# B&R Automation Studio project CleanChemi_SiteManagementSystem (part 3)

#### HA_DirSanitize.st
```iecst
(* Sanitizes File Device *)
FUNCTION_BLOCK HA_DirSanitize
	IF enable = FALSE THEN
		Internal.State										:= DIRSANITIZE_RESET;
	END_IF;

	CASE Internal.State OF
		DIRSANITIZE_RESET:
			status											:= 65534;
			brsmemset(ADR(Internal),0,SIZEOF(Internal));
			Internal.State									:= DIRSANITIZE_IDLE;
		DIRSANITIZE_IDLE:
			status											:= 65534;
			IF enable THEN
				IF pDevice <> 0 AND pDirDef <> 0 AND pFileList <> 0 THEN
					brsmemset(ADR(Internal),0,SIZEOF(Internal));
					status									:= 65535;
					Internal.State							:= DIRSANITIZE_EVALUATE_DIR;
				ELSE
					brsmemset(ADR(Internal),0,SIZEOF(Internal));
					status									:= 60001;
					Internal.State							:= DIRSANITIZE_ERROR;
				END_IF;
			END_IF;
		DIRSANITIZE_EVALUATE_DIR:
			status											:= 65535;
			// Determine DirIdx
			FOR Internal.i := 0 TO MAX_DIR_MAN_FILE_LIST_IDX DO
				brsmemcpy(ADR(Internal.FileListItem),pFileList+SIZEOF(Internal.FileListItem)*Internal.i,SIZEOF(Internal.FileListItem));
				IF Internal.FileListItem.Path = '' AND Internal.FileListItem.IsDir = FALSE THEN
					EXIT;
				ELSE
					Internal.Found 							:= FALSE;
					FOR Internal.j := 0 TO MAX_DIR_DEF_IDX DO
						brsmemcpy(ADR(Internal.DirDefItem),pDirDef+SIZEOF(Internal.DirDefItem)*Internal.j,SIZEOF(Internal.DirDefItem));
						IF Internal.DirDefItem.Valid THEN
							IF Internal.FileListItem.Path = Internal.DirDefItem.DirPath OR Internal.FileListItem.Path = '' THEN
								Internal.FileListItem.DirIdx := Internal.j;
								Internal.Found 				:= TRUE;
								EXIT;
							END_IF;
						END_IF;
					END_FOR;
					IF NOT Internal.Found THEN
						FOR Internal.j := MAX_DIR_DEF_IDX TO 0 BY -1 DO
							brsmemcpy(ADR(Internal.DirDefItem),pDirDef+SIZEOF(Internal.DirDefItem)*Internal.j,SIZEOF(Internal.DirDefItem));
							IF Internal.DirDefItem.Valid THEN
								Internal.Find := FIND(Internal.FileListItem.Path,Internal.DirDefItem.DirPath);
								IF Internal.Find <> 0 THEN
									Internal.TempPath := DELETE(Internal.FileListItem.Path,LEN(Internal.DirDefItem.DirPath),1);
									IF FIND(Internal.TempPath,'/') <> 0 OR Internal.DirDefItem.DirPath = '' THEN
										Internal.FileListItem.DirIdx := Internal.j;
										EXIT;
									END_IF;
								END_IF;
							END_IF;
						END_FOR;
					END_IF;
					brsmemcpy(pFileList+SIZEOF(Internal.FileListItem)*Internal.i,ADR(Internal.FileListItem),SIZEOF(Internal.FileListItem));
				END_IF;
			END_FOR;

			// Handle Directory Sanitation
			Internal.Found									:= FALSE;
			FOR Internal.i := 0 TO MAX_DIR_MAN_FILE_LIST_IDX DO
				brsmemcpy(ADR(Internal.FileListItem),pFileList+SIZEOF(Internal.FileListItem)*Internal.i,SIZEOF(Internal.FileListItem));
				IF Internal.FileListItem.Path = '' AND Internal.FileListItem.IsDir = FALSE THEN
					EXIT;
				ELSIF Internal.FileListItem.IsDir THEN
					brsmemcpy(ADR(Internal.DirDefItem),pDirDef+SIZEOF(Internal.DirDefItem)*Internal.FileListItem.DirIdx,SIZEOF(Internal.DirDefItem));
					IF NOT Internal.DirDefItem.Sanitize.AllowUndefinedDir AND Internal.DirDefItem.DirPath <> Internal.FileListItem.Path THEN
						Internal.Found					:= TRUE;
						Internal.FileListItem.Internal.1 := 1;
						brsmemcpy(pFileList+SIZEOF(Internal.FileListItem)*Internal.i,ADR(Internal.FileListItem),SIZEOF(Internal.FileListItem));
					END_IF;
				END_IF;
			END_FOR;
			Internal.State 									:= DIRSANITIZE_DELETE_DIR_CMD;
		DIRSANITIZE_DELETE_DIR_CMD:
			status											:= 65535;
			Internal.Found									:= FALSE;
			FOR Internal.i := 0 TO MAX_DIR_MAN_FILE_LIST_IDX DO
				brsmemcpy(ADR(Internal.FileListItem),pFileList+SIZEOF(Internal.FileListItem)*Internal.i,SIZEOF(Internal.FileListItem));
				IF Internal.FileListItem.Path = '' AND Internal.FileListItem.IsDir = FALSE THEN
					EXIT;
				ELSIF Internal.FileListItem.IsDir AND Internal.FileListItem.Internal.1 = 1 AND NOT Internal.FileListItem.Internal.2 = 1 THEN
					Internal.Found							:= TRUE;
					EXIT;
				END_IF;
			END_FOR;
			IF Internal.Found THEN
				Internal.DirDeleteEx_0.enable 				:= TRUE;
				Internal.DirDeleteEx_0.pDevice 				:= pDevice;
				Internal.DirDeleteEx_0.pName 				:= ADR(Internal.FileListItem.Path);
				Internal.State 								:= DIRSANITIZE_DELETE_DIR_WAIT;
			ELSE
				Internal.State 								:= DIRSANITIZE_EVALUATE_FILE;
			END_IF;
		DIRSANITIZE_DELETE_DIR_WAIT:
			status											:= 65535;
			IF Internal.DirDeleteEx_0.status = 0 OR (Internal.DirDeleteEx_0.status <> ERR_FUB_BUSY AND Internal.DirDeleteEx_0.status <> ERR_FUB_ENABLE_FALSE) THEN
				Internal.DirDeleteEx_0.enable 				:= FALSE;
				Internal.FileListItem1 						:= Internal.FileListItem;
				FOR Internal.i := 0 TO MAX_DIR_MAN_FILE_LIST_IDX DO
					brsmemcpy(ADR(Internal.FileListItem),pFileList+SIZEOF(Internal.FileListItem)*Internal.i,SIZEOF(Internal.FileListItem));
					IF Internal.FileListItem.Path = '' AND Internal.FileListItem.IsDir = FALSE THEN
						EXIT;
					ELSIF FIND(Internal.FileListItem.Path,Internal.FileListItem1.Path) <> 0 THEN
						Internal.FileListItem.Internal.3 	:= 1;
						brsmemcpy(pFileList+SIZEOF(Internal.FileListItem)*Internal.i,ADR(Internal.FileListItem),SIZEOF(Internal.FileListItem));
					END_IF;
				END_FOR;
				Internal.j 									:= 0;
				FOR Internal.i := 0 TO MAX_DIR_MAN_FILE_LIST_IDX DO
					brsmemcpy(ADR(Internal.FileListItem),pFileList+SIZEOF(Internal.FileListItem)*Internal.i,SIZEOF(Internal.FileListItem));
					IF Internal.FileListItem.Path = '' AND Internal.FileListItem.IsDir = FALSE THEN
						EXIT;
					ELSIF Internal.FileListItem.Internal.3 = 0 THEN
						IF Internal.j <> Internal.i THEN
							Internal.Size						:= (MAX_DIR_MAN_FILE_LIST_IDX+1-Internal.i);
							brsmemmove(pFileList+Internal.j*SIZEOF(Internal.FileListItem),pFileList+Internal.i*SIZEOF(Internal.FileListItem),SIZEOF(Internal.FileListItem)*Internal.Size);
							brsmemset(pFileList+(Internal.j+Internal.Size)*SIZEOF(Internal.FileListItem),0,SIZEOF(Internal.FileListItem)*(Internal.i-Internal.j));
						END_IF;
						Internal.j							:= Internal.j + (Internal.i-Internal.j)+1;
						Internal.i							:= Internal.j-1;
					ELSE
						brsmemset(pFileList+Internal.i*SIZEOF(Internal.FileListItem),0,SIZEOF(Internal.FileListItem));
					END_IF;
				END_FOR;
				Internal.State 								:= DIRSANITIZE_DELETE_DIR_CMD;
			END_IF;
		DIRSANITIZE_EVALUATE_FILE:
			status											:= 65535;

			// Handle File Sanitation By Root
			Internal.Found									:= FALSE;
			FOR Internal.i := 0 TO MAX_DIR_MAN_FILE_LIST_IDX DO
				brsmemcpy(ADR(Internal.FileListItem),pFileList+SIZEOF(Internal.FileListItem)*Internal.i,SIZEOF(Internal.FileListItem));
				IF Internal.FileListItem.Path = '' AND Internal.FileListItem.IsDir = FALSE THEN
					EXIT;
				ELSIF NOT Internal.FileListItem.IsDir THEN
					brsmemcpy(ADR(Internal.DirDefItem),pDirDef+SIZEOF(Internal.DirDefItem)*Internal.FileListItem.DirIdx,SIZEOF(Internal.DirDefItem));
					IF Internal.DirDefItem.Sanitize.SanitizeFilesByRoot THEN
						Internal.TempPath 					:= '';
						brsstrcat(ADR(Internal.TempPath),ADR(Internal.DirDefItem.DirPath));
						brsstrcat(ADR(Internal.TempPath),ADR('/'));
						brsstrcat(ADR(Internal.TempPath),ADR(Internal.DirDefItem.Sanitize.FileRoot));
						IF FIND(Internal.FileListItem.Path,Internal.TempPath) = 0 THEN
							Internal.Found					:= TRUE;
							Internal.FileListItem.Internal.1 := 1;
							brsmemcpy(pFileList+SIZEOF(Internal.FileListItem)*Internal.i,ADR(Internal.FileListItem),SIZEOF(Internal.FileListItem));
						END_IF;
					END_IF;
					IF Internal.DirDefItem.Sanitize.SanitizeFilesByExt THEN
						IF FIND(Internal.FileListItem.Path,Internal.DirDefItem.Sanitize.FileExtension) = 0 THEN
							Internal.Found					:= TRUE;
							Internal.FileListItem.Internal.1 := 1;
							brsmemcpy(pFileList+SIZEOF(Internal.FileListItem)*Internal.i,ADR(Internal.FileListItem),SIZEOF(Internal.FileListItem));
						END_IF;
					END_IF;
				END_IF;
			END_FOR;

			// Check if found in the last step. If so we have to go delete these files before counting them for size and number of files.
			IF Internal.Found THEN
				Internal.State 								:= DIRSANITIZE_DELETE_FILE_CMD;
			ELSE
				// Reorder Files for Evaluation
				FOR Internal.i := 0 TO MAX_DIR_MAN_FILE_LIST_IDX-1 DO
					brsmemcpy(ADR(Internal.FileListItem),pFileList+SIZEOF(Internal.FileListItem)*Internal.i,SIZEOF(Internal.FileListItem));
					brsmemcpy(ADR(Internal.FileListItem1),pFileList+SIZEOF(Internal.FileListItem1)*(Internal.i+1),SIZEOF(Internal.FileListItem1));
					IF (Internal.FileListItem.Path = '' AND Internal.FileListItem.IsDir = FALSE) OR (Internal.FileListItem1.Path = '' AND Internal.FileListItem1.IsDir = FALSE) THEN
						EXIT;
					ELSE
						IF Internal.FileListItem.DirIdx = Internal.FileListItem1.DirIdx THEN
							IF Internal.FileListItem.DateUDINT < Internal.FileListItem1.DateUDINT THEN
								brsmemcpy(pFileList+SIZEOF(Internal.FileListItem1)*Internal.i,ADR(Internal.FileListItem1),SIZEOF(Internal.FileListItem1));
								brsmemcpy(pFileList+SIZEOF(Internal.FileListItem)*(Internal.i+1),ADR(Internal.FileListItem),SIZEOF(Internal.FileListItem));
							END_IF;
						END_IF;
					END_IF;
				END_FOR;
				// Delete Files Based On File Number and Size Restriction
				Internal.Found								:= FALSE;
				Internal.CurrentDirIdx						:= 0;
				Internal.FileCount							:= 1;
				Internal.SizeCount							:= 0;
				FOR Internal.i := 0 TO MAX_DIR_MAN_FILE_LIST_IDX DO
					brsmemcpy(ADR(Internal.FileListItem),pFileList+SIZEOF(Internal.FileListItem)*Internal.i,SIZEOF(Internal.FileListItem));
					IF Internal.FileListItem.Path = '' AND Internal.FileListItem.IsDir = FALSE THEN
						EXIT;
					ELSIF NOT Internal.FileListItem.IsDir THEN
						IF Internal.CurrentDirIdx <> Internal.FileListItem.DirIdx THEN
							Internal.CurrentDirIdx 			:= Internal.FileListItem.DirIdx;
							Internal.FileCount				:= 1;
							Internal.SizeCount				:= Internal.FileListItem.Size;
						ELSE
							Internal.FileCount				:= Internal.FileCount + 1;
							Internal.SizeCount				:= Internal.SizeCount + Internal.FileListItem.Size;
						END_IF;
						brsmemcpy(ADR(Internal.DirDefItem),pDirDef+SIZEOF(Internal.DirDefItem)*Internal.FileListItem.DirIdx,SIZEOF(Internal.DirDefItem));
						IF Internal.FileCount > Internal.DirDefItem.Sanitize.MaxFiles OR Internal.SizeCount > Internal.DirDefItem.Sanitize.MaxSize THEN
							Internal.Found					:= TRUE;
							Internal.FileListItem.Internal.1 := 1;
							brsmemcpy(pFileList+SIZEOF(Internal.FileListItem)*Internal.i,ADR(Internal.FileListItem),SIZEOF(Internal.FileListItem));
						END_IF;
					END_IF;
				END_FOR;
				IF Internal.Found THEN
					Internal.State 							:= DIRSANITIZE_DELETE_FILE_CMD;
				ELSE
					Internal.State 							:= DIRSANITIZE_DONE;
				END_IF;
			END_IF;
		DIRSANITIZE_DELETE_FILE_CMD:
			status											:= 65535;
			Internal.Found									:= FALSE;
			FOR Internal.i := 0 TO MAX_DIR_MAN_FILE_LIST_IDX DO
				brsmemcpy(ADR(Internal.FileListItem),pFileList+SIZEOF(Internal.FileListItem)*Internal.i,SIZEOF(Internal.FileListItem));
				IF Internal.FileListItem.Path = '' AND Internal.FileListItem.IsDir = FALSE THEN
					EXIT;
				ELSIF NOT Internal.FileListItem.IsDir AND Internal.FileListItem.Internal.1 = 1 THEN
					Internal.FileListItem.Internal.1 := 0;
					Internal.FileListItem.Internal.3 := 1;
					brsmemcpy(pFileList+SIZEOF(Internal.FileListItem)*Internal.i,ADR(Internal.FileListItem),SIZEOF(Internal.FileListItem));
					Internal.Found							:= TRUE;
					EXIT;
				END_IF;
			END_FOR;
			IF Internal.Found THEN
				Internal.FileDelete_0.enable 				:= TRUE;
				Internal.FileDelete_0.pDevice 				:= pDevice;
				Internal.FileDelete_0.pName 				:= ADR(Internal.FileListItem.Path);
				Internal.State 								:= DIRSANITIZE_DELETE_FILE_WAIT;
			ELSE
				Internal.State 								:= DIRSANITIZE_EVALUATE_FILE;
			END_IF;
		DIRSANITIZE_DELETE_FILE_WAIT:
			status											:= 65535;
			IF Internal.FileDelete_0.status = 0 OR (Internal.FileDelete_0.status <> ERR_FUB_BUSY AND Internal.FileDelete_0.status <> ERR_FUB_ENABLE_FALSE) THEN
				Internal.FileDelete_0.enable 				:= FALSE;
				Internal.j 									:= 0;
				FOR Internal.i := 0 TO MAX_DIR_MAN_FILE_LIST_IDX DO
					brsmemcpy(ADR(Internal.FileListItem),pFileList+SIZEOF(Internal.FileListItem)*Internal.i,SIZEOF(Internal.FileListItem));
					IF Internal.FileListItem.Path = '' AND Internal.FileListItem.IsDir = FALSE THEN
						EXIT;
					ELSIF Internal.FileListItem.Internal.3 = 0 THEN
						IF Internal.j <> Internal.i THEN
							Internal.Size						:= (MAX_DIR_MAN_FILE_LIST_IDX+1-Internal.i);
							brsmemmove(pFileList+Internal.j*SIZEOF(Internal.FileListItem),pFileList+Internal.i*SIZEOF(Internal.FileListItem),SIZEOF(Internal.FileListItem)*Internal.Size);
							brsmemset(pFileList+(Internal.j+Internal.Size)*SIZEOF(Internal.FileListItem),0,SIZEOF(Internal.FileListItem)*(Internal.i-Internal.j));
						END_IF;
						Internal.j							:= Internal.j + (Internal.i-Internal.j)+1;
						Internal.i							:= Internal.j-1;
					ELSE
						brsmemset(pFileList+Internal.i*SIZEOF(Internal.FileListItem),0,SIZEOF(Internal.FileListItem));
					END_IF;
				END_FOR;
				Internal.State 								:= DIRSANITIZE_DELETE_FILE_CMD;
			END_IF;
		DIRSANITIZE_DONE:
			status											:= 0;
		DIRSANITIZE_ERROR:
			// Error
	END_CASE;

	Internal.FileDelete_0();
	Internal.DirDeleteEx_0();

END_FUNCTION_BLOCK
```

#### HA_Dir_USB_Connect.st
```iecst
// This function only supports a single USB flash drive, additional will be ignored.
// When connected the USB can be accessed using Dev Name 'USB_DEVICE'

FUNCTION_BLOCK HA_Dir_USB_Connect

	IF enable = FALSE OR reset THEN
		Internal.State											:= USB_CONNECT_RESET;
	END_IF;

	CASE Internal.State OF
		USB_CONNECT_RESET:
			status												:= 65534;
			brsmemset(ADR(Internal),0,SIZEOF(Internal));
			connected											:= FALSE;
			Internal.State										:= USB_CONNECT_IDLE;
		USB_CONNECT_IDLE:
			status												:= 65534;
			IF enable THEN
				status											:= 65535;
				Internal.State									:= USB_CONNECT_GET_LIST_CMD;
			END_IF;
		USB_CONNECT_GET_LIST_CMD:
			status												:= 65535;
			Internal.UsbNodeListGet_0.enable 					:= TRUE;
			Internal.UsbNodeListGet_0.pBuffer 					:= ADR(Internal.NodeList);
			Internal.UsbNodeListGet_0.bufferSize 				:= SIZEOF(Internal.NodeList);
			Internal.UsbNodeListGet_0.filterInterfaceClass 		:= 8; // FIND ONLY USB FLASH DRIVES
			Internal.UsbNodeListGet_0.filterInterfaceSubClass 	:= 6; // FIND ONLY USB FLASH DRIVES
			Internal.State 										:= USB_CONNECT_GET_LIST_WAIT;
		USB_CONNECT_GET_LIST_WAIT:
			status												:= 65535;
			IF Internal.UsbNodeListGet_0.status = 0 THEN
				Internal.UsbNodeListGet_0.enable 				:= FALSE;
				Internal.State 									:= USB_CONNECT_GET_NODE_CMD;
			ELSIF Internal.UsbNodeListGet_0.status <> ERR_FUB_BUSY AND Internal.UsbNodeListGet_0.status <> ERR_FUB_ENABLE_FALSE THEN
				IF Internal.UsbNodeListGet_0.status <> asusbERR_USB_NOTFOUND THEN
					Internal.UsbNodeListGet_0.enable 			:= FALSE;
					status										:= Internal.UsbNodeListGet_0.status;
					Internal.State 								:= USB_CONNECT_ERROR;
				ELSE
					Internal.UsbNodeListGet_0.enable 			:= FALSE;
					Internal.State 								:= USB_CONNECT_DELAY;
				END_IF;
			END_IF;
		USB_CONNECT_GET_NODE_CMD:
			status												:= 65535;
			Internal.UsbNodeGet_0.enable 						:= TRUE;
			Internal.UsbNodeGet_0.pBuffer 						:= ADR(Internal.Node);
			Internal.UsbNodeGet_0.bufferSize 					:= SIZEOF(Internal.Node);
			Internal.UsbNodeGet_0.nodeId 						:= Internal.NodeList;
			Internal.State 										:= USB_CONNECT_GET_NODE_WAIT;
		USB_CONNECT_GET_NODE_WAIT:
			status												:= 65535;
			IF Internal.UsbNodeGet_0.status = 0 THEN
				Internal.UsbNodeGet_0.enable 					:= FALSE;
				brsmemset(ADR(Internal.ParString),0,SIZEOF(Internal.ParString));
				brsstrcat(ADR(Internal.ParString),ADR('/DEVICE='));
				brsstrcat(ADR(Internal.ParString), ADR(Internal.Node.ifName));
				Internal.State 									:= USB_CONNECT_DEVLINK_CMD;
			ELSIF Internal.UsbNodeGet_0.status <> ERR_FUB_BUSY AND Internal.UsbNodeGet_0.status <> ERR_FUB_ENABLE_FALSE THEN
				IF Internal.UsbNodeGet_0.status <> asusbERR_USB_NOTFOUND THEN
					Internal.UsbNodeGet_0.enable 				:= FALSE;
					status										:= Internal.UsbNodeGet_0.status;
					Internal.State 								:= USB_CONNECT_ERROR;
				ELSE
					Internal.UsbNodeGet_0.enable 				:= FALSE;
					Internal.State 								:= USB_CONNECT_DELAY;
				END_IF;
			END_IF;
		USB_CONNECT_DEVLINK_CMD:
			status												:= 65535;
			Internal.DevLink_0.enable 							:= TRUE;
			Internal.DevLink_0.pDevice 							:= ADR('USB_DEVICE');
			Internal.DevLink_0.pParam 							:= ADR(Internal.ParString);
			Internal.State 										:= USB_CONNECT_DEVLINK_WAIT;
		USB_CONNECT_DEVLINK_WAIT:
			status												:= 65535;
			IF Internal.DevLink_0.status = 0 THEN
				Internal.DevLink_0.enable 						:= FALSE;
				Internal.Handle									:= Internal.DevLink_0.handle;
				connected										:= FALSE;
				Internal.State 									:= USB_CONNECT_CHECK_CONNECTED;
			ELSIF Internal.DevLink_0.status <> ERR_FUB_BUSY AND Internal.DevLink_0.status <> ERR_FUB_ENABLE_FALSE THEN
				Internal.DevLink_0.enable 						:= FALSE;
				Internal.State 									:= USB_CONNECT_DEVUNLINK_CMD;
			END_IF;
		USB_CONNECT_CHECK_CONNECTED:
			status												:= 65535;
			Internal.UsbMsDeviceReady_0.enable					:= TRUE;
			Internal.UsbMsDeviceReady_0.pIfName					:= ADR(Internal.Node.ifName);
			Internal.State 										:= USB_CONNECT_CONNECTED;
		USB_CONNECT_CONNECTED:
			status												:= 65535;
			IF Internal.UsbMsDeviceReady_0.status = 0 THEN
				connected										:= TRUE;
				Internal.UsbMsDeviceReady_0.enable 				:= FALSE;
				Internal.State 									:= USB_CONNECT_CHECK_CONNECTED;
			ELSIF Internal.UsbMsDeviceReady_0.status <> ERR_FUB_BUSY AND Internal.UsbMsDeviceReady_0.status <> ERR_FUB_ENABLE_FALSE THEN
				Internal.UsbMsDeviceReady_0.enable 				:= FALSE;
				Internal.State 									:= USB_CONNECT_DEVUNLINK_CMD;
			END_IF;
		USB_CONNECT_DEVUNLINK_CMD:
			status												:= 65535;
			Internal.DevUnlink_0.enable 						:= TRUE;
			Internal.DevUnlink_0.handle 						:= Internal.Handle;
			Internal.State 										:= USB_CONNECT_DEVUNLINK_WAIT;
		USB_CONNECT_DEVUNLINK_WAIT:
			status												:= 65535;
			IF Internal.DevUnlink_0.status = 0 OR (Internal.DevUnlink_0.status <> ERR_FUB_BUSY AND Internal.DevUnlink_0.status <> ERR_FUB_ENABLE_FALSE) THEN
				Internal.DevUnlink_0.enable 					:= FALSE;
				Internal.State 									:= USB_CONNECT_DELAY;
			END_IF;
		USB_CONNECT_DELAY:
			status												:= 65535;
			IF Internal.CTON_Delay.Q OR refresh THEN
				refresh 										:= FALSE;
				Internal.CTON_Delay(IN := FALSE);
				Internal.State 									:= USB_CONNECT_GET_LIST_CMD;
			ELSE
				Internal.CTON_Delay(IN := TRUE, PT := REAL_TO_TIME(delay*1000.0));
			END_IF;
 		USB_CONNECT_ERROR:
			connected 											:= FALSE;
	END_CASE;

	Internal.UsbNodeListGet_0();
	Internal.UsbNodeGet_0();
	Internal.DevLink_0();
	Internal.UsbMsDeviceReady_0();
	Internal.DevUnlink_0();

	IF connected THEN
		status													:= 0;
	END_IF;

END_FUNCTION_BLOCK
```

#### HA_Dir_Transfer.st
```iecst
(* Transfer List from Device to Another. Always Overwrites Existing. If either src or dest path includes directories, then the directories need to exist (this will not create them automatically) *)
FUNCTION_BLOCK HA_Dir_Transfer
	IF NOT enable THEN
		Internal.State 											:= TRANSFER_RESET;
	END_IF;

	CASE Internal.State OF
		TRANSFER_RESET:
			status												:= 65534;
			brsmemset(ADR(Internal),0,SIZEOF(Internal));
			Internal.State 										:= TRANSFER_IDLE;
		TRANSFER_IDLE:
			IF enable THEN
				IF pTransferList <> 0 THEN
					status										:= 65535;
					brsmemset(ADR(Internal),0,SIZEOF(Internal));
					Internal.ListIdx		 					:= 0;
					Internal.State 								:= TRANSFER_CHECK_LIST;
				ELSE
					status										:= 60001;
					Internal.State								:= TRANSFER_ERROR;
				END_IF;
			END_IF;
		TRANSFER_CHECK_LIST:
			status												:= 65535;
			IF Internal.ListIdx >= 0 AND Internal.ListIdx <= MAX_TRANSFER_LIST_IDX THEN
				brsmemcpy(ADR(Internal.TransferListItem),pTransferList+SIZEOF(Internal.TransferListItem)*Internal.ListIdx,SIZEOF(Internal.TransferListItem));
				IF Internal.TransferListItem.Valid THEN
					IF Internal.TransferListItem.SrcDelete AND Internal.TransferListItem.NoTransfer THEN
						IF Internal.TransferListItem.IsDir THEN
							Internal.State 						:= TRANSFER_DIR_DELETE_CMD;
						ELSE
							Internal.State 						:= TRANSFER_FILE_DELETE_CMD;
						END_IF;
					ELSIF Internal.TransferListItem.SrcCreateDir THEN
						Internal.State 							:= TRANSFER_DIR_CREATE_CMD;
					ELSIF Internal.TransferListItem.IsDir THEN
						Internal.State 							:= TRANSFER_DIR_COPY_CMD;
					ELSE
						Internal.State 							:= TRANSFER_FILE_COPY_CMD;
					END_IF;
				ELSE
					Internal.State 								:= TRANSFER_DONE;
				END_IF;
			ELSE
				Internal.State 									:= TRANSFER_DONE;
			END_IF;
		TRANSFER_DIR_COPY_CMD:
			status												:= 65535;
			Internal.DirCopy_0.enable 							:= TRUE;
			Internal.DirCopy_0.option 							:= fiOVERWRITE;
			Internal.DirCopy_0.pSrcDev 							:= ADR(Internal.TransferListItem.SrcDev);
			Internal.DirCopy_0.pSrcDir 							:= ADR(Internal.TransferListItem.SrcPath);
			Internal.DirCopy_0.pDestDev 						:= ADR(Internal.TransferListItem.DestDev);
			Internal.DirCopy_0.pDestDir 						:= ADR(Internal.TransferListItem.DestPath);
			Internal.State 										:= TRANSFER_DIR_COPY_WAIT;
		TRANSFER_DIR_COPY_WAIT:
			status												:= 65535;
			IF Internal.TransferListItem.SrcOrDestUSB AND NOT USB_Connected THEN
				Internal.DirCopy_0.enable 						:= FALSE;
				status											:= 65000;
				Internal.State 									:= TRANSFER_ERROR;
			ELSIF Internal.DirCopy_0.status = 0 THEN
				Internal.DirCopy_0.enable 						:= FALSE;
				IF Internal.TransferListItem.SrcDelete THEN
					Internal.State 								:= TRANSFER_DIR_DELETE_CMD;
				ELSE
					Internal.ListIdx							:= Internal.ListIdx + 1;
					Internal.State 								:= TRANSFER_CHECK_LIST;
				END_IF;
			ELSIF Internal.DirCopy_0.status <> ERR_FUB_BUSY AND Internal.DirCopy_0.status <> ERR_FUB_ENABLE_FALSE THEN
				Internal.DirCopy_0.enable 						:= FALSE;
				status											:= Internal.DirCopy_0.status;
				Internal.State 									:= TRANSFER_ERROR;
			END_IF;
		TRANSFER_DIR_DELETE_CMD:
			status												:= 65535;
			Internal.DirDeleteEx_0.enable 						:= TRUE;
			Internal.DirDeleteEx_0.pDevice 						:= ADR(Internal.TransferListItem.SrcDev);
			Internal.DirDeleteEx_0.pName	 					:= ADR(Internal.TransferListItem.SrcPath);
			Internal.State 										:= TRANSFER_DIR_DELETE_WAIT;
		TRANSFER_DIR_DELETE_WAIT:
			status												:= 65535;
			IF Internal.TransferListItem.SrcOrDestUSB AND NOT USB_Connected THEN
				Internal.DirDeleteEx_0.enable 					:= FALSE;
				status											:= 65000;
				Internal.State 									:= TRANSFER_ERROR;
			ELSIF Internal.DirDeleteEx_0.status = 0 THEN
				Internal.DirDeleteEx_0.enable 					:= FALSE;
				Internal.ListIdx								:= Internal.ListIdx + 1;
				Internal.State 									:= TRANSFER_CHECK_LIST;
			ELSIF Internal.DirDeleteEx_0.status <> ERR_FUB_BUSY AND Internal.DirDeleteEx_0.status <> ERR_FUB_ENABLE_FALSE THEN
				Internal.DirDeleteEx_0.enable 					:= FALSE;
				status											:= Internal.DirDeleteEx_0.status;
				Internal.State 									:= TRANSFER_ERROR;
			END_IF;
		TRANSFER_FILE_COPY_CMD:
			status												:= 65535;
			Internal.FileCopy_0.enable 							:= TRUE;
			Internal.FileCopy_0.option 							:= fiOVERWRITE;
			Internal.FileCopy_0.pSrcDev 						:= ADR(Internal.TransferListItem.SrcDev);
			Internal.FileCopy_0.pSrc	 						:= ADR(Internal.TransferListItem.SrcPath);
			Internal.FileCopy_0.pDestDev 						:= ADR(Internal.TransferListItem.DestDev);
			Internal.FileCopy_0.pDest							:= ADR(Internal.TransferListItem.DestPath);
			Internal.State 										:= TRANSFER_FILE_COPY_WAIT;
		TRANSFER_FILE_COPY_WAIT:
			status												:= 65535;
			IF Internal.TransferListItem.SrcOrDestUSB AND NOT USB_Connected THEN
				Internal.FileCopy_0.enable 						:= FALSE;
				status											:= 65000;
				Internal.State 									:= TRANSFER_ERROR;
			ELSIF Internal.FileCopy_0.status = 0 THEN
				Internal.FileCopy_0.enable 						:= FALSE;
				IF Internal.TransferListItem.SrcDelete THEN
					Internal.State 								:= TRANSFER_FILE_DELETE_CMD;
				ELSE
					Internal.ListIdx							:= Internal.ListIdx + 1;
					Internal.State 								:= TRANSFER_CHECK_LIST;
				END_IF;
			ELSIF Internal.FileCopy_0.status <> ERR_FUB_BUSY AND Internal.FileCopy_0.status <> ERR_FUB_ENABLE_FALSE THEN
				Internal.FileCopy_0.enable 						:= FALSE;
				status											:= Internal.FileCopy_0.status;
				Internal.State 									:= TRANSFER_ERROR;
			END_IF;
		TRANSFER_FILE_DELETE_CMD:
			status												:= 65535;
			Internal.FileDelete_0.enable 						:= TRUE;
			Internal.FileDelete_0.pDevice 						:= ADR(Internal.TransferListItem.SrcDev);
			Internal.FileDelete_0.pName	 						:= ADR(Internal.TransferListItem.SrcPath);
			Internal.State 										:= TRANSFER_FILE_DELETE_WAIT;
		TRANSFER_FILE_DELETE_WAIT:
			status												:= 65535;
			IF Internal.TransferListItem.SrcOrDestUSB AND NOT USB_Connected THEN
				Internal.FileDelete_0.enable 					:= FALSE;
				status											:= 65000;
				Internal.State 									:= TRANSFER_ERROR;
			ELSIF Internal.FileDelete_0.status = 0 THEN
				Internal.FileDelete_0.enable 					:= FALSE;
				Internal.ListIdx								:= Internal.ListIdx + 1;
				Internal.State 									:= TRANSFER_CHECK_LIST;
			ELSIF Internal.FileDelete_0.status <> ERR_FUB_BUSY AND Internal.FileDelete_0.status <> ERR_FUB_ENABLE_FALSE THEN
				Internal.FileDelete_0.enable 					:= FALSE;
				status											:= Internal.FileDelete_0.status;
				Internal.State 									:= TRANSFER_ERROR;
			END_IF;
		TRANSFER_DIR_CREATE_CMD:
			status												:= 65535;
			Internal.DirCreate_0.enable 						:= TRUE;
			Internal.DirCreate_0.pDevice 						:= ADR(Internal.TransferListItem.SrcDev);
			Internal.DirCreate_0.pName	 						:= ADR(Internal.TransferListItem.SrcPath);
			Internal.State 										:= TRANSFER_DIR_CREATE_WAIT;
		TRANSFER_DIR_CREATE_WAIT:
			status												:= 65535;
			IF Internal.TransferListItem.SrcOrDestUSB AND NOT USB_Connected THEN
				Internal.DirCreate_0.enable 					:= FALSE;
				status											:= 65000;
				Internal.State 									:= TRANSFER_ERROR;
			ELSIF Internal.DirCreate_0.status = 0 THEN
				Internal.DirCreate_0.enable 					:= FALSE;
				Internal.ListIdx								:= Internal.ListIdx + 1;
				Internal.State 									:= TRANSFER_CHECK_LIST;
			ELSIF Internal.DirCreate_0.status <> ERR_FUB_BUSY AND Internal.DirCreate_0.status <> ERR_FUB_ENABLE_FALSE THEN
				Internal.FileDelete_0.enable 					:= FALSE;
				status											:= Internal.DirCreate_0.status;
				Internal.State 									:= TRANSFER_ERROR;
			END_IF;
		TRANSFER_DONE:
			status												:= 0;
		TRANSFER_ERROR:
			// Error
	END_CASE;

	index 														:= Internal.ListIdx;

	Internal.DirCreate_0();
	Internal.DirCopy_0();
	Internal.FileCopy_0();
	Internal.DirDeleteEx_0();
	Internal.FileDelete_0();

END_FUNCTION_BLOCK
```

#### HA_DirReadAll.st
```iecst
(* Reads Entire File Device *)
FUNCTION_BLOCK HA_DirReadAll
	IF enable = FALSE THEN
		Internal.State														:= DIRREADALL_RESET;
	END_IF;

	CASE Internal.State OF
		DIRREADALL_RESET:
			status															:= 65534;
			brsmemset(ADR(Internal),0,SIZEOF(Internal));
			Internal.State													:= DIRREADALL_IDLE;
		DIRREADALL_IDLE:
			status															:= 65534;
			IF enable THEN
				IF pDevice <> 0 AND pFileList <> 0 THEN
					brsmemset(ADR(Internal),0,SIZEOF(Internal));
					brsmemset(pFileList,0,(SIZEOF(Internal.FileListItem)*(MAX_DIR_MAN_FILE_LIST_IDX+1)));
					Internal.FileListItem.DateUDINT := 0;
					Internal.FileListItem.IsDir := TRUE;
					Internal.FileListItem.Path := '';
					Internal.FileListItem.Size := 0;
					Internal.FileListItem.Internal.0 := 0;
					Internal.FileListIdx									:= 0;
					IF Internal.FileListIdx <= MAX_DIR_MAN_FILE_LIST_IDX THEN
						brsmemcpy(pFileList+SIZEOF(Internal.FileListItem)*Internal.FileListIdx,ADR(Internal.FileListItem),SIZEOF(Internal.FileListItem));
					END_IF;
					Internal.FileListIdx									:= Internal.FileListIdx + 1;
					status													:= 65535;
					Internal.CurrentDirPath									:= '';
					Internal.State											:= DIRREADALL_OPEN_CMD;
				ELSE
					brsmemset(ADR(Internal),0,SIZEOF(Internal));
					status													:= 60001;
					Internal.State											:= DIRREADALL_ERROR;
				END_IF;
			END_IF;
		DIRREADALL_OPEN_CMD:
			status															:= 65535;
			Internal.DirOpen_0.enable 										:= TRUE;
			Internal.DirOpen_0.pDevice 										:= pDevice;
			Internal.DirOpen_0.pName 										:= ADR(Internal.CurrentDirPath);
			Internal.State 													:= DIRREADALL_OPEN_WAIT;
		DIRREADALL_OPEN_WAIT:
			status															:= 65535;
			IF Internal.DirOpen_0.status = 0 THEN
				Internal.DirOpen_0.enable 									:= FALSE;
				Internal.DirIdent 											:= Internal.DirOpen_0.ident;
				Internal.State 												:= DIRREADALL_READ_CMD;
			ELSIF Internal.DirOpen_0.status <> ERR_FUB_BUSY AND Internal.DirOpen_0.status <> ERR_FUB_ENABLE_FALSE THEN
				Internal.DirOpen_0.enable 									:= FALSE;
				status														:= Internal.DirOpen_0.status;
				Internal.State 												:= DIRREADALL_ERROR;
			END_IF;
		DIRREADALL_READ_CMD:
			status															:= 65535;
			brsmemset(ADR(Internal.DirData),0,SIZEOF(Internal.DirData));
			Internal.DirReadEx_0.enable 									:= TRUE;
			Internal.DirReadEx_0.ident 										:= Internal.DirIdent;
			Internal.DirReadEx_0.pData 										:= ADR(Internal.DirData);
			Internal.DirReadEx_0.data_len 									:= SIZEOF(Internal.DirData);
			Internal.State 													:= DIRREADALL_READ_WAIT;
		DIRREADALL_READ_WAIT:
			status															:= 65535;
			IF Internal.DirReadEx_0.status = 0 THEN
				Internal.DirReadEx_0.enable 								:= FALSE;
				brsmemset(ADR(Internal.FileListItem),0,SIZEOF(Internal.FileListItem));
				IF Internal.DirData.Filename[0] <> 46 THEN // check for '.' or '..' and filter out, '.' is decimal 46 in ascii
					IF Internal.CurrentDirPath <> '' THEN
						brsstrcat(ADR(Internal.FileListItem.Path),ADR(Internal.CurrentDirPath));
						brsstrcat(ADR(Internal.FileListItem.Path),ADR('/'));
					END_IF;
					brsstrcat(ADR(Internal.FileListItem.Path),ADR(Internal.DirData.Filename));
					Internal.FileListItem.DateUDINT 						:= DT_TO_UDINT(Internal.DirData.Date);
					Internal.FileListItem.Size 								:= Internal.DirData.Filelength;
					Internal.FileListItem.IsDir 							:= Internal.DirData.Mode = 1;
					Internal.FileListItem.Internal.0						:= Internal.DirData.Mode = 1;
					IF Internal.FileListIdx >= MAX_DIR_MAN_FILE_LIST_IDX THEN
						Internal.State 										:= DIRREADALL_CLOSE_WAIT;
						Internal.DirClose_0.ident 							:= Internal.DirIdent;
						Internal.DirClose_0.enable 							:= TRUE;
					ELSE
						brsmemcpy(pFileList+SIZEOF(Internal.FileListItem)*Internal.FileListIdx,ADR(Internal.FileListItem),SIZEOF(Internal.FileListItem));
						Internal.FileListIdx								:= Internal.FileListIdx + 1;
						Internal.State 										:= DIRREADALL_READ_CMD;
					END_IF;
				ELSE
					Internal.State 											:= DIRREADALL_READ_CMD;
				END_IF;
			ELSIF Internal.DirReadEx_0.status <> ERR_FUB_BUSY AND Internal.DirReadEx_0.status <> ERR_FUB_ENABLE_FALSE THEN
				Internal.DirReadEx_0.enable 								:= FALSE;
				Internal.DirClose_0.ident 									:= Internal.DirIdent;
				Internal.DirClose_0.enable 									:= TRUE;
				Internal.State 												:= DIRREADALL_CLOSE_WAIT;
			END_IF;
		DIRREADALL_CLOSE_WAIT:
			status															:= 65535;
			IF Internal.DirClose_0.status = 0 OR (Internal.DirClose_0.status <> ERR_FUB_BUSY AND Internal.DirClose_0.status <> ERR_FUB_ENABLE_FALSE) THEN
				Internal.DirClose_0.enable 									:= FALSE;
				IF Internal.FileListIdx >= MAX_DIR_MAN_FILE_LIST_IDX THEN
					Internal.State 											:= DIRREADALL_EVALUATE;
				ELSE
					FOR Internal.i := 0 TO MAX_DIR_MAN_FILE_LIST_IDX DO
						brsmemcpy(ADR(Internal.FileListItem),pFileList+SIZEOF(Internal.FileListItem)*Internal.i,SIZEOF(Internal.FileListItem));
						IF Internal.FileListItem.Path = '' AND Internal.FileListItem.IsDir = FALSE THEN
							Internal.State 									:= DIRREADALL_EVALUATE;
							EXIT;
						ELSIF Internal.FileListItem.Internal.0 = 1 THEN
							Internal.CurrentDirPath							:= Internal.FileListItem.Path;
							Internal.FileListItem.Internal.0				:= 0;
							brsmemcpy(pFileList+SIZEOF(Internal.FileListItem)*Internal.i,ADR(Internal.FileListItem),SIZEOF(Internal.FileListItem));
							Internal.State 									:= DIRREADALL_OPEN_CMD;
							EXIT;
						END_IF;
					END_FOR;
				END_IF;
			END_IF;
		DIRREADALL_EVALUATE:
			status															:= 65535;
//			// Build Lists
//			FOR Internal.i := 0 TO MAX_DIR_MAN_FILE_LIST_IDX DO
//				IF Internal.FileList[Internal.i].Path = '' THEN
//					EXIT;
//				ELSIF Internal.FileList[Internal.i].IsDir THEN
//					FileList[Internal.FileListIdx] 							:= Internal.FileList[Internal.i];
//					IF Internal.FileListIdx < MAX_DIR_MAN_FILE_LIST_IDX THEN
//						Internal.FileListIdx								:= Internal.FileListIdx + 1;
//					END_IF;
//				ELSE
//					FileList[Internal.FileListIdx] 							:= Internal.FileList[Internal.i];
//					IF Internal.FileListIdx < MAX_DIR_MAN_FILE_LIST_IDX THEN
//						Internal.FileListIdx								:= Internal.FileListIdx + 1;
//					END_IF;
//				END_IF;
//			END_FOR;
//			FileList 														:= Internal.FileList;
//			Internal.FileListIdx 											:= 0;
			Internal.State 													:= DIRREADALL_DONE;
		DIRREADALL_DONE:
			status															:= 0;
		DIRREADALL_ERROR:
			// Error
	END_CASE;

	Internal.DirOpen_0();
	Internal.DirReadEx_0();
	Internal.DirClose_0();

END_FUNCTION_BLOCK
```

### Library Logical/Libraries/HA_Convert (IEC)

#### Types.typ - Exported data types
```iecst
TYPE
	HA_DT_Parser_Internal_typ : 	STRUCT
		DateTime : DATE_AND_TIME;
		dateTimeStruct : DTStructure;
		year : STRING[4];
		month : STRING[2];
		day : STRING[2];
		hour : STRING[2];
		minute : STRING[2];
		second : STRING[2];
	END_STRUCT;
	HA_DT_Formatter_Internal_typ : 	STRUCT
		dateTimeStruct : DTStructure;
		year : STRING[4];
		month : STRING[2];
		day : STRING[2];
		hour : STRING[2];
		minute : STRING[2];
		second : STRING[2];
		separator : STRING[1];
		c : USINT;
		i : UDINT;
		formatLen : UDINT;
		format : STRING[80];
		output : STRING[80];
		length : UDINT;
	END_STRUCT;
END_TYPE
```

#### HA_Convert.fun - Exported functions and function blocks
```iecst
FUNCTION HA_DT_Parser : BOOL
	VAR_INPUT
		pValueString : UDINT;
		pOutDT : UDINT;
	END_VAR
	VAR
		Internal : HA_DT_Parser_Internal_typ;
	END_VAR
END_FUNCTION

FUNCTION HA_DT_Formatter : BOOL
	VAR_INPUT
		value : DATE_AND_TIME;
		pInFormatString : UDINT; (*Optional*)
		pOutString : UDINT;
		OutStringLength : UDINT;
	END_VAR
	VAR
		Internal : HA_DT_Formatter_Internal_typ;
	END_VAR
END_FUNCTION
```

#### HA_DT_Formatter.st
```iecst
(* Formats DATE_AND_TIME Value into a string *)
FUNCTION HA_DT_Formatter
	HA_DT_Formatter 								:= TRUE;
	IF pOutString = 0 OR OutStringLength = 0 THEN
		HA_DT_Formatter 							:= FALSE;
	ELSE
		HA_DT_Formatter 							:= TRUE;
		Internal.output								:= '';
		Internal.formatLen 							:= brsstrlen(pInFormatString);
		IF pInFormatString = 0 OR Internal.formatLen = 0 OR Internal.formatLen > SIZEOF(Internal.format)-1 THEN
			Internal.format 						:= 'DT#y-m-d-h:M:s';
			Internal.formatLen 						:= brsstrlen(ADR(Internal.format));
		ELSE
			brsstrcpy(ADR(Internal.format),pInFormatString);
			Internal.formatLen 						:= brsstrlen(ADR(Internal.format));
		END_IF;
		DT_TO_DTStructure(value,ADR(Internal.dateTimeStruct));
		Internal.year 								:= UINT_TO_STRING(Internal.dateTimeStruct.year);
		Internal.month 								:= USINT_TO_STRING(Internal.dateTimeStruct.month);
		Internal.day 								:= USINT_TO_STRING(Internal.dateTimeStruct.day);
		Internal.hour 								:= USINT_TO_STRING(Internal.dateTimeStruct.hour);
		Internal.minute 							:= USINT_TO_STRING(Internal.dateTimeStruct.minute);
		Internal.second 							:= USINT_TO_STRING(Internal.dateTimeStruct.second);
		FOR Internal.i := 0 TO Internal.formatLen DO
			brsmemcpy(ADR(Internal.c),ADR(Internal.format)+Internal.i,1);
		    CASE Internal.c OF
		        121: //'y'
					IF Internal.length + 4 >= OutStringLength-1 THEN
						Internal.output 			:= '';
						HA_DT_Formatter 			:= FALSE;
						RETURN;
					ELSE
						Internal.length				:= brsstrcat(ADR(Internal.output),ADR(Internal.year)) - ADR(Internal.output);
					END_IF;
		        109: //'m'
					IF Internal.length + 2 >= OutStringLength-1 THEN
						Internal.output 			:= '';
						HA_DT_Formatter 			:= FALSE;
						RETURN;
					ELSE
						IF Internal.dateTimeStruct.month <= 9 THEN
							brsstrcat(ADR(Internal.output),ADR('0'));
						END_IF;
						Internal.length				:= brsstrcat(ADR(Internal.output),ADR(Internal.month)) - ADR(Internal.output);
					END_IF;
		        100: //'d'
					IF Internal.length + 2 >= OutStringLength-1 THEN
						Internal.output 			:= '';
						HA_DT_Formatter 			:= FALSE;
						RETURN;
					ELSE
						IF Internal.dateTimeStruct.day <= 9 THEN
							brsstrcat(ADR(Internal.output),ADR('0'));
						END_IF;
						Internal.length				:= brsstrcat(ADR(Internal.output),ADR(Internal.day)) - ADR(Internal.output);
					END_IF;
		        104: //'h'
					IF Internal.length + 2 >= OutStringLength-1 THEN
						Internal.output 			:= '';
						HA_DT_Formatter 			:= FALSE;
						RETURN;
					ELSE
						IF Internal.dateTimeStruct.hour <= 9 THEN
							brsstrcat(ADR(Internal.output),ADR('0'));
						END_IF;
						Internal.length				:= brsstrcat(ADR(Internal.output),ADR(Internal.hour)) - ADR(Internal.output);
					END_IF;
		        77: //'M'
					IF Internal.length + 2 >= OutStringLength-1 THEN
						Internal.output 			:= '';
						HA_DT_Formatter 			:= FALSE;
						RETURN;
					ELSE
						IF Internal.dateTimeStruct.minute <= 9 THEN
							brsstrcat(ADR(Internal.output),ADR('0'));
						END_IF;
						Internal.length				:= brsstrcat(ADR(Internal.output),ADR(Internal.minute)) - ADR(Internal.output);
					END_IF;
		        115: //'s'
					IF Internal.length + 2 >= OutStringLength-1 THEN
						Internal.output 			:= '';
						HA_DT_Formatter 			:= FALSE;
						RETURN;
					ELSE
						IF Internal.dateTimeStruct.second <= 9 THEN
							brsstrcat(ADR(Internal.output),ADR('0'));
						END_IF;
						Internal.length				:= brsstrcat(ADR(Internal.output),ADR(Internal.second)) - ADR(Internal.output);
					END_IF;
		        ELSE
					brsmemset(ADR(Internal.separator),0,SIZEOF(Internal.separator));
					brsmemcpy(ADR(Internal.separator),ADR(Internal.c),1);
					IF Internal.length + 1 >= OutStringLength-1 THEN
						Internal.output 			:= '';
						HA_DT_Formatter 			:= FALSE;
						RETURN;
					ELSE
						Internal.length				:= brsstrcat(ADR(Internal.output),ADR(Internal.separator)) - ADR(Internal.output);
					END_IF;
		    END_CASE
		END_FOR;
		IF NOT HA_DT_Formatter THEN
			brsmemset(pOutString,0,OutStringLength);
		ELSE
			brsstrcpy(pOutString,ADR(Internal.output));
		END_IF;
	END_IF;
END_FUNCTION
```

#### HA_DT_Parser.st
```iecst
(* Parses string into DATE_AND_TIME format !!!!!STRING MUST BE IN THE FORM OF DT#yyyy-mm-dd-hh:MM:ss!!!!! all other will fail*)
FUNCTION HA_DT_Parser
	HA_DT_Parser 						:= TRUE;
	IF pOutDT = 0 OR pValueString = 0 THEN
		HA_DT_Parser 					:= FALSE;
	ELSE
		HA_DT_Parser					:= TRUE;
		brsmemset(ADR(Internal),0,SIZEOF(Internal));
		brsmemcpy(ADR(Internal.year),pValueString+3,4);
		brsmemcpy(ADR(Internal.month),pValueString+8,2);
		brsmemcpy(ADR(Internal.day),pValueString+11,2);
		brsmemcpy(ADR(Internal.hour),pValueString+14,2);
		brsmemcpy(ADR(Internal.minute),pValueString+17,2);
		brsmemcpy(ADR(Internal.second),pValueString+20,2);
		Internal.dateTimeStruct.year	:= STRING_TO_UINT(Internal.year);
		Internal.dateTimeStruct.month	:= STRING_TO_USINT(Internal.month);
		Internal.dateTimeStruct.day		:= STRING_TO_USINT(Internal.day);
		Internal.dateTimeStruct.hour	:= STRING_TO_USINT(Internal.hour);
		Internal.dateTimeStruct.minute	:= STRING_TO_USINT(Internal.minute);
		Internal.dateTimeStruct.second	:= STRING_TO_USINT(Internal.second);
		Internal.DateTime := DTStructure_TO_DT(ADR(Internal.dateTimeStruct));
		brsmemcpy(pOutDT,ADR(Internal.DateTime),SIZEOF(Internal.DateTime));
	END_IF;
END_FUNCTION
```

### Library Logical/Libraries/HA_AlarmX (IEC)

#### Types.typ - Exported data types
```iecst
TYPE
	HA_AlarmX_Helper_Internal_typ : 	STRUCT
		Active : BOOL;
		AddText : STRING[1000];
		ArEventLogGetIdent_0 : ArEventLogGetIdent;
		ArEventLogWrite_0 : ArEventLogWrite;
	END_STRUCT;
	HA_ALARMX_ACTION_ENUM :
		(
		HA_ALARMX_ACTION_NONE,
		HA_ALARMX_ACTION_SET,
		HA_ALARMX_ACTION_SET_NO_LOG,
		HA_ALARMX_ACTION_ACK,
		HA_ALARMX_ACTION_ACK_NO_LOG,
		HA_ALARMX_ACTION_LOG_ONLY
		);
	HA_ALARMX_CORE_STATE_ENUM :
		(
		HA_ALARMX_CORE_RESET,
		HA_ALARMX_CORE_IDLE,
		HA_ALARMX_CORE_SET_C,
		HA_ALARMX_CORE_SET_W
		);
	HA_AlarmX_Core_Internal_typ : 	STRUCT
		state : HA_ALARMX_CORE_STATE_ENUM;
		currentAlarm : HA_AlarmX_Core_Buffer_typ;
		tDelay : CTON;
		i : INT;
	END_STRUCT;
	HA_AlarmX_Core_Buffer_typ : 	STRUCT
		name : STRING[MAX_ALARM_NAME_LEN];
		addText : ARRAY[0..HA_ALARMX_MAX_ADD_DATA_IDX]OF STRING[MAX_ALARM_ADD_DATA];
		allowMultiple : BOOL;
	END_STRUCT;
	HA_AlarmX_AlarmExtraData_typ : 	STRUCT
		AddData : ARRAY[0..HA_ALARMX_MAX_ADD_DATA_IDX]OF STRING[MAX_ALARM_ADD_DATA];
	END_STRUCT;
	HA_AlarmX_CfgMod_Internal_typ : 	STRUCT
		MpAlarmXConfigAlarm_0 : MpAlarmXConfigAlarm;
		AlarmCfg : MpAlarmXAlarmConfigType;
		AlarmName : STRING[MAX_ALARM_NAME_LEN];
		i : USINT;
		CTON_Timeout : CTON;
	END_STRUCT;
	HA_AlarmX_BufferInfo_typ : 	STRUCT
		Address : UDINT;
		Size : UDINT;
	END_STRUCT;
	HA_Module_Alarm_Info_typ : 	STRUCT
		ErrorInfo : USINT;
		IgnoreInfo : USINT;
	END_STRUCT;
END_TYPE
```

#### Constants.var - Exported constants
```iecst
VAR CONSTANT
	HA_MODULE_MAX_ALARM : USINT := 6;
	MAX_ALARM_ADD_DATA : UDINT := 255; (*Maximum Length of the extra alarm text*)
	MAX_ALARM_NAME_LEN : UDINT := 255; (*Maximum Length of the alarm name*)
	HA_ALARMX_BUFFER_IDX : UDINT := 255; (*Length of alarm buffer*)
	HA_ALARMX_MAX_ADD_DATA_IDX : USINT := 3;
END_VAR
```

#### HA_AlarmX.fun - Exported functions and function blocks
```iecst
{REDUND_ERROR} FUNCTION HA_AlarmX_Helper : DINT (*Helper Function for Setting and Acknowledging Alarms with User Logger support.*) (*$GROUP=User,$CAT=User,$GROUPICON=User.png,$CATICON=User.png*)
	VAR_INPUT
		MpLink : MpComIdentType;
		AlarmName : STRING[255];
		AlarmAction : HA_ALARMX_ACTION_ENUM;
		LogEventAddText : STRING[255];
		AllowMultiple : BOOL;
	END_VAR
	VAR
		Internal : HA_AlarmX_Helper_Internal_typ;
	END_VAR
END_FUNCTION

{REDUND_ERROR} FUNCTION_BLOCK HA_AlarmXCore (*TODO: Add your comment here*) (*$GROUP=User,$CAT=User,$GROUPICON=User.png,$CATICON=User.png*)
	VAR_INPUT
		enable : BOOL;
		MpLink : MpComIdentType;
		pBuffer : UDINT;
		pOutputData : REFERENCE TO HA_AlarmX_AlarmExtraData_typ;
		delayTime : TIME;
	END_VAR
	VAR
		internal : HA_AlarmX_Core_Internal_typ;
	END_VAR
END_FUNCTION_BLOCK

{REDUND_ERROR} {REDUND_UNREPLICABLE} FUNCTION_BLOCK HA_AlarmX_CfgModule (*Adds the HA default module alarms to the given alarmxcore*) (*$GROUP=User,$CAT=User,$GROUPICON=User.png,$CATICON=User.png*)
	VAR_INPUT
		MpLink : {REDUND_UNREPLICABLE} UDINT;
		Prefix : {REDUND_UNREPLICABLE} STRING[255];
		CodePrefix : {REDUND_UNREPLICABLE} UDINT;
	END_VAR
	VAR
		internal : {REDUND_UNREPLICABLE} HA_AlarmX_CfgMod_Internal_typ;
	END_VAR
	VAR_OUTPUT
		Error : BOOL;
	END_VAR
END_FUNCTION_BLOCK
```

#### HA_AlarmX_Helper.st
```iecst
(* Helper Function for Setting and Acknowledging Alarms with User Logger support. *)
FUNCTION HA_AlarmX_Helper
	HA_AlarmX_Helper 					:= -1;
	brsmemset(ADR(Internal),0,SIZEOF(Internal));
	Internal.ArEventLogGetIdent_0(Execute := FALSE);
	Internal.ArEventLogGetIdent_0(Execute := TRUE, Name := '$$arlogusr');
	Internal.AddText 					:= AlarmName;
	Internal.Active						:= NOT MpAlarmXCheckState(MpLink,AlarmName,mpALARMX_STATE_NONE);

	CASE AlarmAction OF
		HA_ALARMX_ACTION_NONE:
			HA_AlarmX_Helper 			:= 0;
		HA_ALARMX_ACTION_SET:
			HA_AlarmX_Helper 			:= 0;
			IF NOT Internal.Active OR AllowMultiple THEN
				MpAlarmXSet(MpLink,AlarmName);
				brsmemset(ADR(Internal.AddText),0,SIZEOF(Internal.AddText));
				Internal.AddText 	:= AlarmName;
				HA_brsstrcat(ADR(Internal.AddText),ADR(' - Set'),SIZEOF(Internal.AddText));
				IF LogEventAddText <> '' THEN
					HA_brsstrcat(ADR(Internal.AddText),ADR(' - Info: '),SIZEOF(Internal.AddText));
					HA_brsstrcat(ADR(Internal.AddText),ADR(LogEventAddText),SIZEOF(Internal.AddText));
				END_IF;
				Internal.ArEventLogWrite_0(Execute := FALSE);
				Internal.ArEventLogWrite_0(Execute := TRUE, Ident := Internal.ArEventLogGetIdent_0.Ident, EventID := -536870912, OriginRecordID := 0, ObjectID := 'HA_AlarmX_Helper', AddDataSize := brsstrlen(ADR(Internal.AddText)), AddDataFormat := 1, AddData := ADR(Internal.AddText), TimeStamp := 0);
			END_IF;
		HA_ALARMX_ACTION_SET_NO_LOG:
			HA_AlarmX_Helper 			:= 0;
			IF NOT Internal.Active OR AllowMultiple THEN
				MpAlarmXSet(MpLink,AlarmName);
				brsmemset(ADR(Internal.AddText),0,SIZEOF(Internal.AddText));
			END_IF;
		HA_ALARMX_ACTION_ACK:
			HA_AlarmX_Helper 			:= 0;
			IF Internal.Active THEN
				MpAlarmXAcknowledge(MpLink,AlarmName);
				brsmemset(ADR(Internal.AddText),0,SIZEOF(Internal.AddText));
				Internal.AddText 	:= AlarmName;
				HA_brsstrcat(ADR(Internal.AddText),ADR(' - Ack'),SIZEOF(Internal.AddText));
				IF LogEventAddText <> '' THEN
					HA_brsstrcat(ADR(Internal.AddText),ADR(' - Info: '),SIZEOF(Internal.AddText));
					HA_brsstrcat(ADR(Internal.AddText),ADR(LogEventAddText),SIZEOF(Internal.AddText));
				END_IF;
				Internal.ArEventLogWrite_0(Execute := FALSE);
				Internal.ArEventLogWrite_0(Execute := TRUE, Ident := Internal.ArEventLogGetIdent_0.Ident, EventID := -536870912, OriginRecordID := 0, ObjectID := 'HA_AlarmX_Helper', AddDataSize := brsstrlen(ADR(Internal.AddText)), AddDataFormat := 1, AddData := ADR(Internal.AddText), TimeStamp := 0);
			END_IF;
		HA_ALARMX_ACTION_ACK_NO_LOG:
			HA_AlarmX_Helper 			:= 0;
			IF Internal.Active THEN
				MpAlarmXAcknowledge(MpLink,AlarmName);
			END_IF;
		HA_ALARMX_ACTION_LOG_ONLY:
			HA_AlarmX_Helper 			:= 0;
			brsmemset(ADR(Internal.AddText),0,SIZEOF(Internal.AddText));
			IF LogEventAddText <> '' THEN
				HA_brsstrcat(ADR(Internal.AddText),ADR('Info: '),SIZEOF(Internal.AddText));
				HA_brsstrcat(ADR(Internal.AddText),ADR(LogEventAddText),SIZEOF(Internal.AddText));
				Internal.ArEventLogWrite_0(Execute := FALSE);
				Internal.ArEventLogWrite_0(Execute := TRUE, Ident := Internal.ArEventLogGetIdent_0.Ident, EventID := -536870912, OriginRecordID := 0, ObjectID := 'HA_AlarmX_Helper', AddDataSize := brsstrlen(ADR(Internal.AddText)), AddDataFormat := 1, AddData := ADR(Internal.AddText), TimeStamp := 0);
			END_IF;
	END_CASE;

END_FUNCTION
```

#### HA_AlarmXCore.st
```iecst
(* Alarm Core to handle setting multiple alarms in one cycle with different texts *)
FUNCTION_BLOCK HA_AlarmXCore

	IF enable = FALSE THEN
		internal.state := HA_ALARMX_CORE_RESET;
	END_IF

	CASE internal.state OF

		HA_ALARMX_CORE_RESET:

			brsmemset(ADR(internal.currentAlarm), 0, SIZEOF(internal.currentAlarm));
			internal.state := HA_ALARMX_CORE_IDLE;

		HA_ALARMX_CORE_IDLE:

			IF HA_Array_PeekBtm(pBuffer, SIZEOF(internal.currentAlarm) * HA_ALARMX_BUFFER_IDX, ADR(internal.currentAlarm), SIZEOF(internal.currentAlarm)) > 0 THEN
				HA_Array_Dequeue(pBuffer, SIZEOF(internal.currentAlarm) * HA_ALARMX_BUFFER_IDX, ADR(internal.currentAlarm), SIZEOF(internal.currentAlarm));
				internal.state := HA_ALARMX_CORE_SET_C;
			END_IF

		HA_ALARMX_CORE_SET_C:

			FOR internal.i := 0 TO HA_ALARMX_MAX_ADD_DATA_IDX DO
				pOutputData.AddData[internal.i]	:= internal.currentAlarm.addText[internal.i];
			END_FOR
			HA_AlarmX_Helper(MpLink, internal.currentAlarm.name, HA_ALARMX_ACTION_SET, '', internal.currentAlarm.allowMultiple);

			internal.state := HA_ALARMX_CORE_SET_W;

		HA_ALARMX_CORE_SET_W:

			internal.tDelay.IN	:= TRUE;
			internal.tDelay.PT	:= delayTime;

			IF internal.tDelay.Q THEN
				internal.tDelay.IN	:= FALSE;
				internal.state 		:= HA_ALARMX_CORE_IDLE;
			END_IF

	END_CASE

	internal.tDelay();

END_FUNCTION_BLOCK
```

#### HA_AlarmX_CfgModule.st
```iecst
(* Adds the HA default module alarms to the given alarmxcore *)
FUNCTION_BLOCK HA_AlarmX_CfgModule

	WHILE internal.i < HA_MODULE_MAX_ALARM + 1 DO

		CASE internal.i OF

			0:
				internal.AlarmName														:= Prefix;
				HA_brsstrcat(ADR(internal.AlarmName), ADR('UnhandledCmd'), SIZEOF(internal.AlarmName));
				internal.AlarmCfg.Message												:= '{$$IAT/Alarm.';
				HA_brsstrcat(ADR(internal.AlarmCfg.Message), ADR(internal.AlarmName), SIZEOF(internal.AlarmCfg.Message));
				HA_brsstrcat(ADR(internal.AlarmCfg.Message), ADR('}'), SIZEOF(internal.AlarmCfg.Message));
				internal.AlarmCfg.Code													:= CodePrefix;
				internal.AlarmCfg.Severity												:= 4;
				internal.AlarmCfg.Behavior.AutoReset									:= TRUE;
				internal.AlarmCfg.Behavior.Acknowledge 									:= mpALARMX_ACK_REQ;
				internal.AlarmCfg.Behavior.MultipleInstances 							:= TRUE;
				internal.AlarmCfg.Behavior.ReactionUntilAcknowledged					:= TRUE;
				internal.AlarmCfg.Behavior.HistoryReport.InactiveToActive 				:= TRUE;
				internal.AlarmCfg.Behavior.HistoryReport.UnacknowledgedToAcknowledged	:= TRUE;

			1:
				internal.AlarmName															:= Prefix;
				HA_brsstrcat(ADR(internal.AlarmName), ADR('Severity1'), SIZEOF(internal.AlarmName));
				internal.AlarmCfg.Message												:= '{$$IAT/Alarm.';
				HA_brsstrcat(ADR(internal.AlarmCfg.Message), ADR('Severity1'), SIZEOF(internal.AlarmCfg.Message));
				HA_brsstrcat(ADR(internal.AlarmCfg.Message), ADR('}'), SIZEOF(internal.AlarmCfg.Message));
				internal.AlarmCfg.Code													:= CodePrefix;
				internal.AlarmCfg.Severity												:= 1;
				internal.AlarmCfg.Behavior.AutoReset									:= TRUE;
				internal.AlarmCfg.Behavior.Acknowledge 									:= mpALARMX_ACK_REQ;
				internal.AlarmCfg.Behavior.MultipleInstances 							:= TRUE;
				internal.AlarmCfg.Behavior.ReactionUntilAcknowledged					:= TRUE;
				internal.AlarmCfg.Behavior.HistoryReport.InactiveToActive 				:= TRUE;
				internal.AlarmCfg.Behavior.HistoryReport.UnacknowledgedToAcknowledged	:= TRUE;

			2:
				internal.AlarmName															:= Prefix;
				HA_brsstrcat(ADR(internal.AlarmName), ADR('Severity2'), SIZEOF(internal.AlarmName));
				internal.AlarmCfg.Message												:= '{$$IAT/Alarm.';
				HA_brsstrcat(ADR(internal.AlarmCfg.Message), ADR('Severity2'), SIZEOF(internal.AlarmCfg.Message));
				HA_brsstrcat(ADR(internal.AlarmCfg.Message), ADR('}'), SIZEOF(internal.AlarmCfg.Message));
				internal.AlarmCfg.Code													:= CodePrefix;
				internal.AlarmCfg.Severity												:= 2;
				internal.AlarmCfg.Behavior.AutoReset									:= TRUE;
				internal.AlarmCfg.Behavior.Acknowledge 									:= mpALARMX_ACK_REQ;
				internal.AlarmCfg.Behavior.MultipleInstances 							:= TRUE;
				internal.AlarmCfg.Behavior.ReactionUntilAcknowledged					:= TRUE;
				internal.AlarmCfg.Behavior.HistoryReport.InactiveToActive 				:= TRUE;
				internal.AlarmCfg.Behavior.HistoryReport.UnacknowledgedToAcknowledged	:= TRUE;

			3:
				internal.AlarmName															:= Prefix;
				HA_brsstrcat(ADR(internal.AlarmName), ADR('Severity3'), SIZEOF(internal.AlarmName));
				internal.AlarmCfg.Message												:= '{$$IAT/Alarm.';
				HA_brsstrcat(ADR(internal.AlarmCfg.Message), ADR('Severity3'), SIZEOF(internal.AlarmCfg.Message));
				HA_brsstrcat(ADR(internal.AlarmCfg.Message), ADR('}'), SIZEOF(internal.AlarmCfg.Message));
				internal.AlarmCfg.Code													:= CodePrefix;
				internal.AlarmCfg.Severity												:= 3;
				internal.AlarmCfg.Behavior.AutoReset									:= TRUE;
				internal.AlarmCfg.Behavior.Acknowledge 									:= mpALARMX_ACK_REQ;
				internal.AlarmCfg.Behavior.MultipleInstances 							:= TRUE;
				internal.AlarmCfg.Behavior.ReactionUntilAcknowledged					:= TRUE;
				internal.AlarmCfg.Behavior.HistoryReport.InactiveToActive 				:= TRUE;
				internal.AlarmCfg.Behavior.HistoryReport.UnacknowledgedToAcknowledged	:= TRUE;

			4:
				internal.AlarmName															:= Prefix;
				HA_brsstrcat(ADR(internal.AlarmName), ADR('Severity4'), SIZEOF(internal.AlarmName));
				internal.AlarmCfg.Message												:= '{$$IAT/Alarm.';
				HA_brsstrcat(ADR(internal.AlarmCfg.Message), ADR('Severity4'), SIZEOF(internal.AlarmCfg.Message));
				HA_brsstrcat(ADR(internal.AlarmCfg.Message), ADR('}'), SIZEOF(internal.AlarmCfg.Message));
				internal.AlarmCfg.Code													:= CodePrefix;
				internal.AlarmCfg.Severity												:= 4;
				internal.AlarmCfg.Behavior.AutoReset									:= TRUE;
				internal.AlarmCfg.Behavior.Acknowledge 									:= mpALARMX_ACK_REQ;
				internal.AlarmCfg.Behavior.MultipleInstances 							:= TRUE;
				internal.AlarmCfg.Behavior.ReactionUntilAcknowledged					:= TRUE;
				internal.AlarmCfg.Behavior.HistoryReport.InactiveToActive 				:= TRUE;
				internal.AlarmCfg.Behavior.HistoryReport.UnacknowledgedToAcknowledged	:= TRUE;

			5:
				internal.AlarmName															:= Prefix;
				HA_brsstrcat(ADR(internal.AlarmName), ADR('Severity5'), SIZEOF(internal.AlarmName));
				internal.AlarmCfg.Message												:= '{$$IAT/Alarm.';
				HA_brsstrcat(ADR(internal.AlarmCfg.Message), ADR('Severity5'), SIZEOF(internal.AlarmCfg.Message));
				HA_brsstrcat(ADR(internal.AlarmCfg.Message), ADR('}'), SIZEOF(internal.AlarmCfg.Message));
				internal.AlarmCfg.Code													:= CodePrefix;
				internal.AlarmCfg.Severity												:= 5;
				internal.AlarmCfg.Behavior.AutoReset									:= TRUE;
				internal.AlarmCfg.Behavior.Acknowledge 									:= mpALARMX_ACK_REQ;
				internal.AlarmCfg.Behavior.MultipleInstances 							:= TRUE;
				internal.AlarmCfg.Behavior.ReactionUntilAcknowledged					:= TRUE;
				internal.AlarmCfg.Behavior.HistoryReport.InactiveToActive 				:= TRUE;
				internal.AlarmCfg.Behavior.HistoryReport.UnacknowledgedToAcknowledged	:= TRUE;

			6:
				internal.AlarmName														:= Prefix;
				HA_brsstrcat(ADR(internal.AlarmName), ADR('CmdIgnored'), SIZEOF(internal.AlarmName));
				internal.AlarmCfg.Message												:= '{$$IAT/Alarm.';
				HA_brsstrcat(ADR(internal.AlarmCfg.Message), ADR(internal.AlarmName), SIZEOF(internal.AlarmCfg.Message));
				HA_brsstrcat(ADR(internal.AlarmCfg.Message), ADR('}'), SIZEOF(internal.AlarmCfg.Message));
				internal.AlarmCfg.Code													:= CodePrefix + 6;
				internal.AlarmCfg.Severity												:= 0;
				internal.AlarmCfg.Behavior.AutoReset									:= TRUE;
				internal.AlarmCfg.Behavior.Acknowledge 									:= mpALARMX_ACK_REQ;
				internal.AlarmCfg.Behavior.MultipleInstances 							:= TRUE;
				internal.AlarmCfg.Behavior.ReactionUntilAcknowledged					:= TRUE;
				internal.AlarmCfg.Behavior.HistoryReport.InactiveToActive 				:= TRUE;
				internal.AlarmCfg.Behavior.HistoryReport.UnacknowledgedToAcknowledged	:= TRUE;

		END_CASE

		internal.MpAlarmXConfigAlarm_0.MpLink			:= MpLink;
		internal.MpAlarmXConfigAlarm_0.Enable			:= TRUE;
		internal.MpAlarmXConfigAlarm_0.Name				:= ADR(internal.AlarmName);
		internal.MpAlarmXConfigAlarm_0.Configuration	:= ADR(internal.AlarmCfg);
		internal.MpAlarmXConfigAlarm_0.Save				:= TRUE;

		IF internal.MpAlarmXConfigAlarm_0.CommandDone THEN
			internal.i := internal.i + 1;
			internal.MpAlarmXConfigAlarm_0.Save := FALSE;
		ELSIF internal.MpAlarmXConfigAlarm_0.Error THEN
			Error	:= TRUE;
			RETURN;
		END_IF;

		internal.MpAlarmXConfigAlarm_0();
	END_WHILE

END_FUNCTION_BLOCK
```

### Library Logical/Libraries/HA_ItemX (IEC)

#### Types.typ - Exported data types
```iecst
TYPE
	ItemX_typ : 	STRUCT
		CurrentUID : UDINT; (*REQUIRED*)
		ValidIndex : BOOL; (*REQUIRED*)
		ReturnedIndex : INT; (*REQUIRED*)
		Elem : ItemX_Elem_typ; (*REQUIRED*)
		List : ARRAY[0..MAX_ITEM_X_IDX]OF ItemX_Elem_typ; (*REQUIRED*)
	END_STRUCT;
	ItemX_Elem_typ : 	STRUCT
		UID : UDINT; (*REQUIRED*)
		State : ITEM_X_STATE_ENUM; (*REQUIRED*)
		LastLoc : ITEM_X_LOC_ENUM; (*REQUIRED*)
		Loc : ITEM_X_LOC_ENUM; (*REQUIRED*)
		Par : ItemX_Par_typ; (*REQUIRED*)
		Status : ItemX_Status_typ; (*REQUIRED*)
	END_STRUCT;
	ItemX_Status_typ : 	STRUCT
		Position : REAL;
		Length : REAL;
		ManuallyRemoved : BOOL;
		Rejected : BOOL;
		Passed : BOOL;
		TimeIn : DATE_AND_TIME;
		TimeOut : DATE_AND_TIME;
		Error : BOOL;
	END_STRUCT;
	ItemX_Par_typ : 	STRUCT
		ProductID : INT;
		Recipe : ItemX_Par_Recipe_typ;
	END_STRUCT;
	ItemX_Par_Recipe_typ : 	STRUCT
		MaxLength : REAL;
	END_STRUCT;
	ITEM_X_STATE_ENUM :
		(
		ITEM_X_STATE_UNDEFINED, (*REQUIRED*)
		ITEM_X_STATE_WAIT_START,
		ITEM_X_STATE_ACTIVE,
		ITEM_X_STATE_DONE,
		ITEM_X_STATE_UNKNOWN,
		ITEM_X_STATE_ERRORSTOP
		);
	ITEM_X_LOC_ENUM :
		(
		ITEM_X_LOC_UNDEFINED, (*REQUIRED*)
		ITEM_X_LOC_UNKNOWN
		);
	HA_ItemX_Internal_typ : 	STRUCT
		i : INT;
		j : INT;
		tempItemX : ItemX_Elem_typ;
		tempIndex : INT;
		tempUID : UDINT;
	END_STRUCT;
END_TYPE
```

#### Constants.var - Exported constants
```iecst
VAR CONSTANT
	MAX_ITEM_X_IDX : INT := 15;
	MAX_NAME_STRING_LENGTH : INT := 30;
END_VAR
```

#### HA_ItemX.fun - Exported functions and function blocks
```iecst
{REDUND_ERROR} FUNCTION HA_ItemX_DeleteByIndex : BOOL (* *) (*$GROUP=User,$CAT=User,$GROUPICON=User.png,$CATICON=User.png*)
	VAR_INPUT
		Index : INT;
	END_VAR
	VAR_IN_OUT
		ItemX : ItemX_typ;
	END_VAR
	VAR
		Internal : HA_ItemX_Internal_typ;
	END_VAR
END_FUNCTION

{REDUND_ERROR} FUNCTION HA_ItemX_DeleteByUID : BOOL (* *) (*$GROUP=User,$CAT=User,$GROUPICON=User.png,$CATICON=User.png*)
	VAR_INPUT
		UID : UDINT;
	END_VAR
	VAR_IN_OUT
		ItemX : ItemX_typ;
	END_VAR
	VAR
		Internal : HA_ItemX_Internal_typ;
	END_VAR
END_FUNCTION

{REDUND_ERROR} FUNCTION HA_ItemX_UID_TO_Index : BOOL (* *) (*$GROUP=User,$CAT=User,$GROUPICON=User.png,$CATICON=User.png*)
	VAR_INPUT
		UID : UDINT;
	END_VAR
	VAR_IN_OUT
		ItemX : ItemX_typ;
	END_VAR
	VAR
		Internal : HA_ItemX_Internal_typ;
	END_VAR
END_FUNCTION

{REDUND_ERROR} FUNCTION HA_ItemX_Sanitize : BOOL (* *) (*$GROUP=User,$CAT=User,$GROUPICON=User.png,$CATICON=User.png*)
	VAR_IN_OUT
		ItemX : ItemX_typ;
	END_VAR
	VAR
		Internal : HA_ItemX_Internal_typ;
	END_VAR
END_FUNCTION

{REDUND_ERROR} FUNCTION HA_ItemX_Reorder_LowToHighUID : BOOL (* *) (*$GROUP=User,$CAT=User,$GROUPICON=User.png,$CATICON=User.png*)
	VAR_IN_OUT
		ItemX : ItemX_typ;
	END_VAR
	VAR
		Internal : HA_ItemX_Internal_typ;
	END_VAR
END_FUNCTION

{REDUND_ERROR} FUNCTION HA_ItemX_Reorder_HighToLowUID : BOOL (* *) (*$GROUP=User,$CAT=User,$GROUPICON=User.png,$CATICON=User.png*)
	VAR_IN_OUT
		ItemX : ItemX_typ;
	END_VAR
	VAR
		Internal : HA_ItemX_Internal_typ;
	END_VAR
END_FUNCTION

{REDUND_ERROR} FUNCTION HA_ItemX_IndexLowestUID : BOOL (* *) (*$GROUP=User,$CAT=User,$GROUPICON=User.png,$CATICON=User.png*)
	VAR_IN_OUT
		ItemX : ItemX_typ;
	END_VAR
	VAR
		Internal : HA_ItemX_Internal_typ;
	END_VAR
END_FUNCTION

{REDUND_ERROR} FUNCTION HA_ItemX_IndexHighestUID : BOOL (* *) (*$GROUP=User,$CAT=User,$GROUPICON=User.png,$CATICON=User.png*)
	VAR_IN_OUT
		ItemX : ItemX_typ;
	END_VAR
	VAR
		Internal : HA_ItemX_Internal_typ;
	END_VAR
END_FUNCTION

{REDUND_ERROR} FUNCTION HA_ItemX_FirstOpenIndex : BOOL (* *) (*$GROUP=User,$CAT=User,$GROUPICON=User.png,$CATICON=User.png*)
	VAR_IN_OUT
		ItemX : ItemX_typ;
	END_VAR
	VAR
		Internal : HA_ItemX_Internal_typ;
	END_VAR
END_FUNCTION

{REDUND_ERROR} FUNCTION HA_ItemX_GetElemByIndex : BOOL (* *) (*$GROUP=User,$CAT=User,$GROUPICON=User.png,$CATICON=User.png*)
	VAR_INPUT
		Index : INT;
	END_VAR
	VAR_IN_OUT
		ItemX : ItemX_typ;
	END_VAR
	VAR
		Internal : HA_ItemX_Internal_typ;
	END_VAR
END_FUNCTION

{REDUND_ERROR} FUNCTION HA_ItemX_GetElemByUID : BOOL (* *) (*$GROUP=User,$CAT=User,$GROUPICON=User.png,$CATICON=User.png*)
	VAR_INPUT
		UID : UDINT;
	END_VAR
	VAR_IN_OUT
		ItemX : ItemX_typ;
	END_VAR
	VAR
		Internal : HA_ItemX_Internal_typ;
	END_VAR
END_FUNCTION

{REDUND_ERROR} FUNCTION HA_ItemX_ModElemByIndex : BOOL (* *) (*$GROUP=User,$CAT=User,$GROUPICON=User.png,$CATICON=User.png*)
	VAR_INPUT
		Index : INT;
	END_VAR
	VAR_IN_OUT
		ItemX : ItemX_typ;
	END_VAR
	VAR
		Internal : HA_ItemX_Internal_typ;
	END_VAR
END_FUNCTION

{REDUND_ERROR} FUNCTION HA_ItemX_ModElemByUID : BOOL (* *) (*$GROUP=User,$CAT=User,$GROUPICON=User.png,$CATICON=User.png*)
	VAR_INPUT
		UID : UDINT;
	END_VAR
	VAR_IN_OUT
		ItemX : ItemX_typ;
	END_VAR
	VAR
		Internal : HA_ItemX_Internal_typ;
	END_VAR
END_FUNCTION

{REDUND_ERROR} FUNCTION HA_ItemX_AddElem : BOOL (* *) (*$GROUP=User,$CAT=User,$GROUPICON=User.png,$CATICON=User.png*)
	VAR_IN_OUT
		ItemX : ItemX_typ;
	END_VAR
	VAR
		Internal : HA_ItemX_Internal_typ;
	END_VAR
END_FUNCTION

{REDUND_ERROR} FUNCTION HA_ItemX_IncrementUID : BOOL (* *) (*$GROUP=User,$CAT=User,$GROUPICON=User.png,$CATICON=User.png*)
	VAR_IN_OUT
		ItemX : ItemX_typ;
	END_VAR
	VAR
		Internal : HA_ItemX_Internal_typ;
	END_VAR
END_FUNCTION
```

#### HA_ItemX_FirstOpenIndex.st
```iecst
(* Finds the first open index of the item array *)
FUNCTION HA_ItemX_FirstOpenIndex
	HA_ItemX_FirstOpenIndex							:= FALSE;
	ItemX.ReturnedIndex								:= -1;
	FOR Internal.i := 0 TO MAX_ITEM_X_IDX DO
		IF ItemX.List[Internal.i].UID = 0 THEN
			HA_ItemX_FirstOpenIndex					:= TRUE;
			ItemX.ReturnedIndex						:= Internal.i;
			EXIT;
		END_IF;
	END_FOR;

	// This is here for keeping the ItemX structure up to date and should be at the bottom of every function call in the library
	ItemX.ValidIndex									:= FALSE;
	IF ItemX.ReturnedIndex >= 0 AND ItemX.ReturnedIndex <= MAX_ITEM_X_IDX THEN
		ItemX.ValidIndex								:= TRUE;
	END_IF;

END_FUNCTION
```

#### HA_ItemX_UID_TO_Index.st
```iecst
(* Returns the first index matching the UID entered *)
FUNCTION HA_ItemX_UID_TO_Index
	HA_ItemX_UID_TO_Index							:= FALSE;
	ItemX.ReturnedIndex								:= -1;
	FOR Internal.i := 0 TO MAX_ITEM_X_IDX DO
		IF ItemX.List[Internal.i].UID = UID THEN
			HA_ItemX_UID_TO_Index					:= TRUE;
			ItemX.ReturnedIndex						:= Internal.i;
			EXIT;
		END_IF;
	END_FOR;

	// This is here for keeping the ItemX structure up to date and should be at the bottom of every function call in the library
	ItemX.ValidIndex									:= FALSE;
	IF ItemX.ReturnedIndex >= 0 AND ItemX.ReturnedIndex <= MAX_ITEM_X_IDX THEN
		ItemX.ValidIndex								:= TRUE;
	END_IF;

END_FUNCTION
```

#### HA_ItemX_DeleteByUID.st
```iecst
(* Deletes the first index matching the UID entered, Returns True if Deleted, False if not found *)
FUNCTION HA_ItemX_DeleteByUID
	HA_ItemX_DeleteByUID								:= FALSE;
	ItemX.ReturnedIndex								:= -1;
	FOR Internal.i := 0 TO MAX_ITEM_X_IDX DO
		IF ItemX.List[Internal.i].UID = UID THEN
			brsmemset(ADR(ItemX.List[Internal.i]),0,SIZEOF(ItemX.List[Internal.i]));
			ItemX.ReturnedIndex						:= Internal.i;
			HA_ItemX_DeleteByUID						:= TRUE;
			EXIT;
		END_IF;
	END_FOR;

	// This is here for keeping the ItemX structure up to date and should be at the bottom of every function call in the library
	ItemX.ValidIndex									:= FALSE;
	IF ItemX.ReturnedIndex >= 0 AND ItemX.ReturnedIndex <= MAX_ITEM_X_IDX THEN
		ItemX.ValidIndex								:= TRUE;
	END_IF;

END_FUNCTION
```

#### HA_ItemX_DeleteByIndex.st
```iecst
(* Deletes the index entered, Returns True if Deleted, False if not in range *)
FUNCTION HA_ItemX_DeleteByIndex
	Internal.i 											:= 0; // This is to avoid a compiler warning that internal is not used.
	HA_ItemX_DeleteByIndex								:= FALSE;
	ItemX.ReturnedIndex									:= -1;
	IF Index >= 0 AND Index <= MAX_ITEM_X_IDX THEN
		brsmemset(ADR(ItemX.List[Index]),0,SIZEOF(ItemX.List[Index]));
		ItemX.ReturnedIndex								:= Index;
		HA_ItemX_DeleteByIndex							:= TRUE;
	END_IF;

	// This is here for keeping the ItemX structure up to date and should be at the bottom of every function call in the library
	ItemX.ValidIndex									:= FALSE;
	IF ItemX.ReturnedIndex >= 0 AND ItemX.ReturnedIndex <= MAX_ITEM_X_IDX THEN
		ItemX.ValidIndex								:= TRUE;
	END_IF;

END_FUNCTION
```

#### HA_ItemX_IndexLowestUID.st
```iecst
(* Returns the index of the lowest UID found in the item array,*)
FUNCTION HA_ItemX_IndexLowestUID
	HA_ItemX_IndexLowestUID							:= FALSE;
	ItemX.ReturnedIndex								:= -1;
	Internal.tempUID								:= 4294967295; // Set to UDINT max
	FOR Internal.i := 0 TO MAX_ITEM_X_IDX DO
		IF ItemX.List[Internal.i].UID < Internal.tempUID AND ItemX.List[Internal.i].UID > 0 THEN
			Internal.tempUID						:= ItemX.List[Internal.i].UID;
			ItemX.ReturnedIndex						:= Internal.i;
			HA_ItemX_IndexLowestUID					:= TRUE;
		END_IF;
	END_FOR;

	// This is here for keeping the ItemX structure up to date and should be at the bottom of every function call in the library
	ItemX.ValidIndex									:= FALSE;
	IF ItemX.ReturnedIndex >= 0 AND ItemX.ReturnedIndex <= MAX_ITEM_X_IDX THEN
		ItemX.ValidIndex								:= TRUE;
	END_IF;

END_FUNCTION
```

#### HA_ItemX_IndexHighestUID.st
```iecst
(* Returns the index of the highest UID found in the item array, -1 if All UID are 0 *)
FUNCTION HA_ItemX_IndexHighestUID
	HA_ItemX_IndexHighestUID							:= FALSE;
	ItemX.ReturnedIndex								:= -1;
	Internal.tempUID								:= 0;
	FOR Internal.i := 0 TO MAX_ITEM_X_IDX DO
		IF ItemX.List[Internal.i].UID > Internal.tempUID THEN
			Internal.tempUID						:= ItemX.List[Internal.i].UID;
			ItemX.ReturnedIndex						:= Internal.i;
			HA_ItemX_IndexHighestUID					:= TRUE;
		END_IF;
	END_FOR;

	// This is here for keeping the ItemX structure up to date and should be at the bottom of every function call in the library
	ItemX.ValidIndex									:= FALSE;
	IF ItemX.ReturnedIndex >= 0 AND ItemX.ReturnedIndex <= MAX_ITEM_X_IDX THEN
		ItemX.ValidIndex								:= TRUE;
	END_IF;

END_FUNCTION
```

#### HA_ItemX_Reorder_HighToLowUID.st
```iecst
(* Reorders the array to be from high to low in terms of UID *)
FUNCTION HA_ItemX_Reorder_HighToLowUID
	HA_ItemX_Reorder_HighToLowUID					:= TRUE;
	FOR Internal.i := 0 TO MAX_ITEM_X_IDX DO
		// Find Next Highest Index
		Internal.tempIndex							:= Internal.i;
		FOR Internal.j := Internal.i TO MAX_ITEM_X_IDX DO
			IF ItemX.List[Internal.j].UID > ItemX.List[Internal.tempIndex].UID THEN
				Internal.tempIndex					:= Internal.j;
			END_IF;
		END_FOR;
		// Swap ItemXs
		Internal.tempItemX							:= ItemX.List[Internal.i];
		ItemX.List[Internal.i]						:= ItemX.List[Internal.tempIndex];
		ItemX.List[Internal.tempIndex]				:= Internal.tempItemX;
		IF ItemX.List[Internal.i].UID = 0 THEN
			ItemX.ReturnedIndex 						:= Internal.i;
			EXIT;
		END_IF;
	END_FOR;

	// This is here for keeping the ItemX structure up to date and should be at the bottom of every function call in the library
	ItemX.ValidIndex									:= FALSE;
	IF ItemX.ReturnedIndex >= 0 AND ItemX.ReturnedIndex <= MAX_ITEM_X_IDX THEN
		ItemX.ValidIndex								:= TRUE;
	END_IF;

END_FUNCTION
```

#### HA_ItemX_Reorder_LowToHighUID.st
```iecst
(* Reorders the array to be from low to high in terms of UID, 0 elements left at the end of the array *)
FUNCTION HA_ItemX_Reorder_LowToHighUID
	HA_ItemX_Reorder_LowToHighUID					:= TRUE;
	FOR Internal.i := 0 TO MAX_ITEM_X_IDX DO
		// Find Next Lowest Index
		Internal.tempIndex							:= Internal.i;
		IF ItemX.List[Internal.tempIndex].UID = 0 THEN
			Internal.tempUID						:= 4294967295; // Set to UDINT max
		ELSE
			Internal.tempUID						:= ItemX.List[Internal.tempIndex].UID;
		END_IF;
		FOR Internal.j := Internal.i TO MAX_ITEM_X_IDX DO
			IF ItemX.List[Internal.j].UID < Internal.tempUID AND ItemX.List[Internal.j].UID > 0 THEN
				Internal.tempIndex					:= Internal.j;
				Internal.tempUID					:= ItemX.List[Internal.tempIndex].UID;
			END_IF;
		END_FOR;
		// Swap ItemXs
		Internal.tempItemX							:= ItemX.List[Internal.i];
		ItemX.List[Internal.i]						:= ItemX.List[Internal.tempIndex];
		ItemX.List[Internal.tempIndex]				:= Internal.tempItemX;
		IF ItemX.List[Internal.i].UID = 0 THEN
			ItemX.ReturnedIndex 						:= Internal.i;
			EXIT;
		END_IF;
	END_FOR;

	// This is here for keeping the ItemX structure up to date and should be at the bottom of every function call in the library
	ItemX.ValidIndex									:= FALSE;
	IF ItemX.ReturnedIndex >= 0 AND ItemX.ReturnedIndex <= MAX_ITEM_X_IDX THEN
		ItemX.ValidIndex								:= TRUE;
	END_IF;

END_FUNCTION
```

#### HA_ItemX_Sanitize.st
```iecst
(* Deletes all ItemXs that have UID of 0 *)
FUNCTION HA_ItemX_Sanitize
	HA_ItemX_Sanitize								:= TRUE;
	FOR Internal.i := 0 TO MAX_ITEM_X_IDX DO
		IF ItemX.List[Internal.i].UID = 0 THEN
			brsmemset(ADR(ItemX.List[Internal.i]),0,SIZEOF(ItemX.List[Internal.i]));
		END_IF;
	END_FOR;

	HA_ItemX_FirstOpenIndex(ItemX);
	// This is here for keeping the ItemX structure up to date and should be at the bottom of every function call in the library
	ItemX.ValidIndex									:= FALSE;
	IF ItemX.ReturnedIndex >= 0 AND ItemX.ReturnedIndex <= MAX_ITEM_X_IDX THEN
		ItemX.ValidIndex								:= TRUE;
	END_IF;

END_FUNCTION
```

#### HA_ItemX_IncrementUID.st
```iecst
(* IncrementsUID, Ensures that the UID will be the Highest in the list if it isnt *)
FUNCTION HA_ItemX_IncrementUID
	HA_ItemX_IncrementUID							:= TRUE;
	ItemX.CurrentUID								:= ItemX.CurrentUID + 1;

	Internal.tempUID								:= 0;
	FOR Internal.i := 0 TO MAX_ITEM_X_IDX DO
		IF ItemX.List[Internal.i].UID > Internal.tempUID THEN
			Internal.tempUID						:= ItemX.List[Internal.i].UID;
		END_IF;
	END_FOR;
	IF Internal.tempUID >= ItemX.CurrentUID THEN
		ItemX.CurrentUID							:= Internal.tempUID + 1;
	END_IF;

	// This is here for keeping the ItemX structure up to date and should be at the bottom of every function call in the library
	ItemX.ValidIndex								:= FALSE;
	IF ItemX.ReturnedIndex >= 0 AND ItemX.ReturnedIndex <= MAX_ITEM_X_IDX THEN
		ItemX.ValidIndex							:= TRUE;
	END_IF;

END_FUNCTION
```

#### HA_ItemX_AddElem.st
```iecst
(* Adds Elem to List, returns true if successful and changes index to where it was added *)
FUNCTION HA_ItemX_AddElem

	HA_ItemX_AddElem								:= FALSE;
	ItemX.ReturnedIndex								:= -1;
	FOR Internal.i := 0 TO MAX_ITEM_X_IDX DO
		IF ItemX.List[Internal.i].UID = 0 THEN
			HA_ItemX_AddElem						:= TRUE;
			ItemX.ReturnedIndex						:= Internal.i;
			HA_ItemX_IncrementUID(ItemX);
			ItemX.Elem.UID							:= ItemX.CurrentUID;
			ItemX.List[Internal.i]					:= ItemX.Elem;
			EXIT;
		END_IF;
	END_FOR;

	// This is here for keeping the ItemX structure up to date and should be at the bottom of every function call in the library
	ItemX.ValidIndex								:= FALSE;
	IF ItemX.ReturnedIndex >= 0 AND ItemX.ReturnedIndex <= MAX_ITEM_X_IDX THEN
		ItemX.ValidIndex							:= TRUE;
	END_IF;

END_FUNCTION
```

#### HA_ItemX_ModElemByUID.st
```iecst
(* Modifies Elem in List without changing UID, returns true if successful *)
FUNCTION HA_ItemX_ModElemByUID

	HA_ItemX_ModElemByUID							:= FALSE;
	ItemX.ReturnedIndex								:= -1;

	FOR Internal.i := 0 TO MAX_ITEM_X_IDX DO
		IF ItemX.List[Internal.i].UID = UID THEN
			ItemX.Elem.UID							:= UID;
			ItemX.List[Internal.i]					:= ItemX.Elem;
			ItemX.List[Internal.i].UID 				:= UID;
			ItemX.ReturnedIndex						:= Internal.i;
			HA_ItemX_ModElemByUID					:= TRUE;
			EXIT;
		END_IF;
	END_FOR;

	// This is here for keeping the ItemX structure up to date and should be at the bottom of every function call in the library
	ItemX.ValidIndex								:= FALSE;
	IF ItemX.ReturnedIndex >= 0 AND ItemX.ReturnedIndex <= MAX_ITEM_X_IDX THEN
		ItemX.ValidIndex							:= TRUE;
	END_IF;

END_FUNCTION
```

#### HA_ItemX_ModElemByIndex.st
```iecst
(* Modifies Elem in List without changing UID, returns true if successful *)
FUNCTION HA_ItemX_ModElemByIndex

	HA_ItemX_ModElemByIndex							:= FALSE;
	ItemX.ReturnedIndex								:= -1;

	IF Index >= 0 AND Index <= MAX_ITEM_X_IDX THEN
		IF ItemX.List[Index].UID = 0 THEN
			HA_ItemX_AddElem(ItemX);
		ELSE
			Internal.tempUID						:= ItemX.List[Index].UID;
			ItemX.List[Index]						:= ItemX.Elem;
			ItemX.List[Internal.i].UID 				:= Internal.tempUID;
		END_IF;
		ItemX.ReturnedIndex							:= Index;
		HA_ItemX_ModElemByIndex						:= TRUE;
	END_IF;

	// This is here for keeping the ItemX structure up to date and should be at the bottom of every function call in the library
	ItemX.ValidIndex								:= FALSE;
	IF ItemX.ReturnedIndex >= 0 AND ItemX.ReturnedIndex <= MAX_ITEM_X_IDX THEN
		ItemX.ValidIndex							:= TRUE;
	END_IF;

END_FUNCTION
```

#### HA_ItemX_GetElemByUID.st
```iecst
(* Gets Elem in List, returns true if successful *)
FUNCTION HA_ItemX_GetElemByUID

	HA_ItemX_GetElemByUID							:= FALSE;
	ItemX.ReturnedIndex								:= -1;

	FOR Internal.i := 0 TO MAX_ITEM_X_IDX DO
		IF ItemX.List[Internal.i].UID = UID THEN
			ItemX.Elem								:= ItemX.List[Internal.i];
			ItemX.ReturnedIndex						:= Internal.i;
			HA_ItemX_GetElemByUID					:= TRUE;
			EXIT;
		END_IF;
	END_FOR;

	// This is here for keeping the ItemX structure up to date and should be at the bottom of every function call in the library
	ItemX.ValidIndex								:= FALSE;
	IF ItemX.ReturnedIndex >= 0 AND ItemX.ReturnedIndex <= MAX_ITEM_X_IDX THEN
		ItemX.ValidIndex							:= TRUE;
	END_IF;

END_FUNCTION
```

#### HA_ItemX_GetElemByIndex.st
```iecst
(* Gets Elem in List, returns true if successful *)
FUNCTION HA_ItemX_GetElemByIndex
	Internal.i 										:= 0; // This is to avoid a compiler warning that internal is not used.
	HA_ItemX_GetElemByIndex							:= FALSE;
	ItemX.ReturnedIndex								:= -1;

	IF Index >= 0 AND Index <= MAX_ITEM_X_IDX THEN
		IF ItemX.List[Index].UID <> 0 THEN
			ItemX.Elem								:= ItemX.List[Index];
			ItemX.ReturnedIndex						:= Index;
			HA_ItemX_GetElemByIndex					:= TRUE;
		END_IF;
	END_IF;

	// This is here for keeping the ItemX structure up to date and should be at the bottom of every function call in the library
	ItemX.ValidIndex								:= FALSE;
	IF ItemX.ReturnedIndex >= 0 AND ItemX.ReturnedIndex <= MAX_ITEM_X_IDX THEN
		ItemX.ValidIndex							:= TRUE;
	END_IF;

END_FUNCTION
```

### Library Logical/Libraries/HA_RAND (ANSIC, version 1.00.0)

#### HA_RAND.fun - Exported functions and function blocks
```iecst
{REDUND_ERROR} FUNCTION SRAND : BOOL (*seed function*) (*$GROUP=User,$CAT=User,$GROUPICON=User.png,$CATICON=User.png*)
	VAR_INPUT
		Seed : UINT;
	END_VAR
END_FUNCTION

{REDUND_ERROR} FUNCTION DRAND : DINT (*Generates random number between (low,high)*) (*$GROUP=User,$CAT=User,$GROUPICON=User.png,$CATICON=User.png*)
	VAR_INPUT
		Low : DINT;
		High : DINT;
	END_VAR
END_FUNCTION

{REDUND_ERROR} FUNCTION RRAND : LREAL (*Generates random number between (low,high)*) (*$GROUP=User,$CAT=User,$GROUPICON=User.png,$CATICON=User.png*)
	VAR_INPUT
		Low : LREAL;
		High : LREAL;
	END_VAR
END_FUNCTION

{REDUND_ERROR} FUNCTION RAND : INT (*Generates random number*) (*$GROUP=User,$CAT=User,$GROUPICON=User.png,$CATICON=User.png*)
END_FUNCTION
```

#### SRAND.c
```c
#include <bur/plctypes.h>
#include <stdlib.h>
#ifdef __cplusplus
	extern "C"
	{
#endif
	#include "HA_RAND.h"
#ifdef __cplusplus
	};
#endif
/* seed function */
plcbit SRAND(unsigned short Seed)
{
	srand(Seed);
	return 1;
}
```

#### RAND.c
```c
#include <bur/plctypes.h>
#include <stdlib.h>
#ifdef __cplusplus
	extern "C"
	{
#endif
	#include "HA_RAND.h"
#ifdef __cplusplus
	};
#endif
/* Generates random number */
signed short RAND(void)
{
	return (signed short)rand();
}
```

#### RRAND.c
```c
#include <bur/plctypes.h>
#include <stdlib.h>
#ifdef __cplusplus
	extern "C"
	{
#endif
	#include "HA_RAND.h"
#ifdef __cplusplus
	};
#endif
/* Generates random number between the (low,high) */
double RRAND(double low, double high)
{
	return (((double)rand())/2147483647.0)*(high-low)+low;
}
```

#### DRAND.c
```c
#include <bur/plctypes.h>
#include <stdlib.h>
#ifdef __cplusplus
	extern "C"
	{
#endif
	#include "HA_RAND.h"
#ifdef __cplusplus
	};
#endif
/* Generates random number between the (low,high) */
signed long DRAND(signed long low, signed long high)
{
	return (rand() % (high - low + 1)) + low;
}
```

### Library Logical/Libraries/HA_Array (IEC)
Depends on: AsBrStr

#### Constants.var - Exported constants
```iecst
VAR CONSTANT
	HA_ARRAY_MAXELEMENTSIZE : UINT := 2000;
END_VAR
```

#### HA_Array.fun - Exported functions and function blocks
```iecst
{REDUND_ERROR} FUNCTION HA_Array_PeekTop : INT (*Peeks at the top index of an array without removing it*) (*$GROUP=User,$CAT=User,$GROUPICON=User.png,$CATICON=User.png*)
	VAR_INPUT
		pBuffer : UDINT;
		sizeBuffer : UDINT;
		pElement : UDINT;
		SizeElement : UDINT;
	END_VAR
	VAR
		emptyData : ARRAY[0..HA_ARRAY_MAXELEMENTSIZE] OF USINT;
		i : UDINT;
	END_VAR
END_FUNCTION

{REDUND_ERROR} FUNCTION HA_Array_AddTop : INT (*Adds the first index of an array*) (*$GROUP=User,$CAT=User,$GROUPICON=User.png,$CATICON=User.png*)
	VAR_INPUT
		pBuffer : UDINT;
		SizeBuffer : UDINT;
		pElement : UDINT;
		SizeElement : UDINT;
	END_VAR
END_FUNCTION

{REDUND_ERROR} FUNCTION HA_Array_AddBottom : BOOL (*Removes the last index of an array*) (*$GROUP=User,$CAT=User,$GROUPICON=User.png,$CATICON=User.png*)
	VAR_INPUT
		pBuffer : UDINT;
		SizeBuffer : UDINT;
		pElement : UDINT;
		SizeElement : UDINT;
	END_VAR
END_FUNCTION

{REDUND_ERROR} FUNCTION HA_Array_PeekBtm : INT (*Copies the last index in an array to the output without removing it*) (*$GROUP=User,$CAT=User,$GROUPICON=User.png,$CATICON=User.png*)
	VAR_INPUT
		pBuffer : UDINT;
		sizeBuffer : UDINT;
		pElement : UDINT;
		SizeElement : UDINT;
	END_VAR
	VAR
		emptyData : ARRAY[0..HA_ARRAY_MAXELEMENTSIZE] OF USINT;
		i : DINT;
	END_VAR
END_FUNCTION

{REDUND_ERROR} FUNCTION HA_Array_Pop : INT (*Pops the top index out of the array into out variable*) (*$GROUP=User,$CAT=User,$GROUPICON=User.png,$CATICON=User.png*)
	VAR_INPUT
		pBuffer : UDINT;
		sizeBuffer : UDINT;
		pElement : UDINT;
		SizeElement : UDINT;
	END_VAR
	VAR
		emptyData : ARRAY[0..HA_ARRAY_MAXELEMENTSIZE] OF USINT;
		i : UDINT;
		nextSpot : UDINT;
	END_VAR
END_FUNCTION

{REDUND_ERROR} FUNCTION HA_Array_Dequeue : INT (*Dequeues the last index in an array to the output*) (*$GROUP=User,$CAT=User,$GROUPICON=User.png,$CATICON=User.png*)
	VAR_INPUT
		pBuffer : UDINT;
		sizeBuffer : UDINT;
		pElement : UDINT;
		SizeElement : UDINT;
	END_VAR
	VAR
		emptyData : ARRAY[0..HA_ARRAY_MAXELEMENTSIZE] OF USINT;
		i : DINT;
	END_VAR
END_FUNCTION

{REDUND_ERROR} FUNCTION HA_Array_Pack : INT (*TODO: Add your comment here*) (*$GROUP=User,$CAT=User,$GROUPICON=User.png,$CATICON=User.png*)
	VAR_INPUT
		pBuffer : UDINT;
		sizeBuffer : UDINT;
		SizeElement : UDINT;
	END_VAR
	VAR
		emptyData : ARRAY[0..HA_ARRAY_MAXELEMENTSIZE] OF USINT;
		i : UDINT;
		dataFound : UDINT;
	END_VAR
END_FUNCTION
```

#### HA_Array_AddTop.st
```iecst
(* Adds the first index of an array *)
FUNCTION HA_Array_AddTop

	HA_Array_AddTop := 0;

	//Input Error Checking
	IF 	pBuffer = 0 THEN
		HA_Array_AddTop.15 := 1;
		HA_Array_AddTop.0  := 1;
	END_IF

	IF pElement = 0 THEN
		HA_Array_AddTop.15 := 1;
		HA_Array_AddTop.1  := 1;
	END_IF

	IF SizeBuffer = 0 THEN
		HA_Array_AddTop.15 := 1;
		HA_Array_AddTop.2  := 1;
	END_IF

	IF SizeElement = 0 THEN
		HA_Array_AddTop.15 := 1;
		HA_Array_AddTop.3  := 1;
	END_IF

	IF SizeBuffer < SizeElement * 2 THEN
		HA_Array_AddTop.15 := 1;
		HA_Array_AddTop.4  := 1;
	END_IF

	IF SizeBuffer MOD SizeElement <> 0 THEN
		HA_Array_AddTop.15 := 1;
		HA_Array_AddTop.5  := 1;
	END_IF

	IF HA_Array_AddTop = 0 THEN
		//Everything passed we can go to work
		brsmemmove(pBuffer + SizeElement, pBuffer, SizeBuffer - SizeElement);
		brsmemcpy(pBuffer, pElement, SizeElement);
	END_IF

END_FUNCTION
```

#### HA_Array_AddBottom.st
```iecst
(* Removes the last index of an array *)
FUNCTION HA_Array_AddBottom
	pBuffer;
	SizeBuffer;
	pElement;
	SizeElement;
	HA_Array_AddBottom := TRUE;
END_FUNCTION
```

#### HA_Array_PeekTop.st
```iecst
(* Peeks at the top index of an array without removing it *)
FUNCTION HA_Array_PeekTop

	HA_Array_PeekTop := 0;
	brsmemset(ADR(emptyData), 0, SIZEOF(emptyData));

	//Validate input parameters
	IF pBuffer = 0 THEN
		HA_Array_PeekTop.0  := TRUE;
		HA_Array_PeekTop.15 := TRUE;
	END_IF

	IF sizeBuffer = 0 THEN
		HA_Array_PeekTop.1  := TRUE;
		HA_Array_PeekTop.15 := TRUE;
	END_IF

	IF pElement = 0 THEN
		HA_Array_PeekTop.2  := TRUE;
		HA_Array_PeekTop.15 := TRUE;
	END_IF

	IF SizeElement = 0 THEN
		HA_Array_PeekTop.3  := TRUE;
		HA_Array_PeekTop.15 := TRUE;
	END_IF

	IF sizeBuffer MOD SizeElement <> 0 THEN
		HA_Array_PeekTop.4  := TRUE;
		HA_Array_PeekTop.15 := TRUE;
	END_IF

	IF SizeElement > HA_ARRAY_MAXELEMENTSIZE THEN
		HA_Array_PeekTop.5  := TRUE;
		HA_Array_PeekTop.15 := TRUE;
	END_IF

	//Everything passed we can go a head and peek
	IF HA_Array_PeekTop = 0 THEN
		FOR i:=0 TO (sizeBuffer / SizeElement)-1 DO
			IF brsmemcmp(pBuffer + SizeElement*i, ADR(emptyData), SizeElement) <> 0 THEN
				//We found the first index
				brsmemcpy(pElement, pBuffer + SizeElement*i, SizeElement);
				HA_Array_PeekTop := 1;
				EXIT;
			END_IF
		END_FOR
	END_IF

END_FUNCTION
```

#### HA_Array_PeekBtm.st
```iecst
(*Peeks at the bottom of the array without moving it.. cheeky monkey
	Returns (-) number for error, 0 for nothing in array and 1 when it finds something*)
FUNCTION HA_Array_PeekBtm

	HA_Array_PeekBtm := 0;
	brsmemset(ADR(emptyData), 0, SIZEOF(emptyData));

	//Validate input parameters
	IF pBuffer = 0 THEN
		HA_Array_PeekBtm.0  := TRUE;
		HA_Array_PeekBtm.15 := TRUE;
	END_IF

	IF sizeBuffer = 0 THEN
		HA_Array_PeekBtm.1  := TRUE;
		HA_Array_PeekBtm.15 := TRUE;
	END_IF

	IF pElement = 0 THEN
		HA_Array_PeekBtm.2  := TRUE;
		HA_Array_PeekBtm.15 := TRUE;
	END_IF

	IF SizeElement = 0 THEN
		HA_Array_PeekBtm.3  := TRUE;
		HA_Array_PeekBtm.15 := TRUE;
	END_IF

	IF sizeBuffer MOD SizeElement <> 0 THEN
		HA_Array_PeekBtm.4  := TRUE;
		HA_Array_PeekBtm.15 := TRUE;
	END_IF

	IF SizeElement > HA_ARRAY_MAXELEMENTSIZE THEN
		HA_Array_PeekBtm.5  := TRUE;
		HA_Array_PeekBtm.15 := TRUE;
	END_IF

	//Everything passed we can go a head and peek
	IF HA_Array_PeekBtm = 0 THEN
		FOR i:= (sizeBuffer / SizeElement)-1 TO 0 BY -1 DO
			IF brsmemcmp(pBuffer + SizeElement*DINT_TO_UDINT(i), ADR(emptyData), SizeElement) <> 0 THEN
				//We found the first index
				brsmemcpy(pElement, pBuffer + SizeElement*DINT_TO_UDINT(i), SizeElement);
				HA_Array_PeekBtm := 1;
				EXIT;
			END_IF
		END_FOR
	END_IF

END_FUNCTION
```

#### HA_Array_Pop.st
```iecst
(* Pops the top index out of the array into out variable *)
FUNCTION HA_Array_Pop

	HA_Array_Pop := 0;
	brsmemset(ADR(emptyData), 0, SIZEOF(emptyData));

	//Validate input parameters
	IF pBuffer = 0 THEN
		HA_Array_Pop.0  := TRUE;
		HA_Array_Pop.15 := TRUE;
	END_IF

	IF sizeBuffer = 0 THEN
		HA_Array_Pop.1  := TRUE;
		HA_Array_Pop.15 := TRUE;
	END_IF

	IF pElement = 0 THEN
		HA_Array_Pop.2  := TRUE;
		HA_Array_Pop.15 := TRUE;
	END_IF

	IF SizeElement = 0 THEN
		HA_Array_Pop.3  := TRUE;
		HA_Array_Pop.15 := TRUE;
	END_IF

	IF sizeBuffer MOD SizeElement <> 0 THEN
		HA_Array_Pop.4  := TRUE;
		HA_Array_Pop.15 := TRUE;
	END_IF

	IF SizeElement > HA_ARRAY_MAXELEMENTSIZE THEN
		HA_Array_Pop.5  := TRUE;
		HA_Array_Pop.15 := TRUE;
	END_IF

	//Everything passed we can go a head and look for an index to pop
	IF HA_Array_Pop = 0 THEN
		FOR i:=0 TO (sizeBuffer / SizeElement) - 1 DO
			IF brsmemcmp(pBuffer + SizeElement*i, ADR(emptyData), SizeElement) <> 0 THEN
				//We found the first index
				brsmemcpy(pElement, pBuffer + SizeElement*i, SizeElement);
				nextSpot := brsmemmove(pBuffer, pBuffer + SizeElement*(i+1), sizeBuffer - SizeElement * (i+1));
				brsmemset(nextSpot, 0, SizeElement*(i+1));
				HA_Array_Pop := 1;
				EXIT;
			END_IF
		END_FOR
	END_IF

END_FUNCTION
```

#### HA_Array_Dequeue.st
```iecst
(* Dequeues the last index in an array to the output *)
FUNCTION HA_Array_Dequeue

	HA_Array_Dequeue := 0;
	brsmemset(ADR(emptyData), 0, SIZEOF(emptyData));

	//Validate input parameters
	IF pBuffer = 0 THEN
		HA_Array_Dequeue.0  := TRUE;
		HA_Array_Dequeue.15 := TRUE;
	END_IF

	IF sizeBuffer = 0 THEN
		HA_Array_Dequeue.1  := TRUE;
		HA_Array_Dequeue.15 := TRUE;
	END_IF

	IF pElement = 0 THEN
		HA_Array_Dequeue.2  := TRUE;
		HA_Array_Dequeue.15 := TRUE;
	END_IF

	IF SizeElement = 0 THEN
		HA_Array_Dequeue.3  := TRUE;
		HA_Array_Dequeue.15 := TRUE;
	END_IF

	IF sizeBuffer MOD SizeElement <> 0 THEN
		HA_Array_Dequeue.4  := TRUE;
		HA_Array_Dequeue.15 := TRUE;
	END_IF

	IF SizeElement > HA_ARRAY_MAXELEMENTSIZE THEN
		HA_Array_Dequeue.5  := TRUE;
		HA_Array_Dequeue.15 := TRUE;
	END_IF

	//Everything passed we can go a head and peek
	IF HA_Array_Dequeue = 0 THEN
		FOR i:= (sizeBuffer / SizeElement) - 1 TO 0 BY -1 DO
			IF brsmemcmp(pBuffer + SizeElement*DINT_TO_UDINT(i), ADR(emptyData), SizeElement) <> 0 THEN
				//We found the first index
				brsmemcpy(pElement, pBuffer + SizeElement*DINT_TO_UDINT(i), SizeElement);
				brsmemset(pBuffer + SizeElement*DINT_TO_UDINT(i), 0, SizeElement);
				HA_Array_Dequeue := 1;
				EXIT;
			END_IF
		END_FOR
	END_IF

END_FUNCTION
```

#### HA_Array_Pack.st
```iecst
(* TODO: Actually make this work *)
FUNCTION HA_Array_Pack

	HA_Array_Pack := 0;
	brsmemset(ADR(emptyData), 0, SIZEOF(emptyData));

	//Validate input parameters
	IF pBuffer = 0 THEN
		HA_Array_Pack.0  := TRUE;
		HA_Array_Pack.15 := TRUE;
	END_IF

	IF sizeBuffer = 0 THEN
		HA_Array_Pack.1  := TRUE;
		HA_Array_Pack.15 := TRUE;
	END_IF

	IF HA_Array_Pack = 0 THEN
		FOR i:= (sizeBuffer / SizeElement) TO 1 BY -1 DO
			IF brsmemcmp(pBuffer + SizeElement*i, ADR(emptyData), SizeElement) = 0 THEN
				IF dataFound <> 0 THEN
					brsmemmove(pBuffer + SizeElement*i, pBuffer + SizeElement*(i+1), dataFound*SizeElement);
				END_IF
			ELSE
				dataFound := dataFound + 1;
			END_IF
		END_FOR
	END_IF

END_FUNCTION
```

### Library Logical/Libraries/HA_SysErr (IEC, version 1.00.0)
Depends on: ArTextSys, AsBrStr, ArEventLog

#### Types.typ - Exported data types
```iecst
TYPE
	Internal_HA_SysErr_Log : 	STRUCT
		State : INT;
		HA_SysErr_Lookup_0 : HA_SysErr_Lookup;
		ArEventLogGetIdent_0 : ArEventLogGetIdent;
		ArEventLogWrite_0 : ArEventLogWrite;
		AddData : STRING[255];
	END_STRUCT;
	Internal_HA_SysErr_Lookup : 	STRUCT
		ArTextSysGetText_0 : ArTextSysGetText;
		TextID : STRING[255];
		ErrorNumString : STRING[80];
		State : INT;
	END_STRUCT;
END_TYPE
```

#### HA_SysErr.fun - Exported functions and function blocks
```iecst
{REDUND_ERROR} FUNCTION_BLOCK HA_SysErr_Lookup (*Returns System Error If It Exists In Table*) (*$GROUP=User,$CAT=User,$GROUPICON=User.png,$CATICON=User.png*)
	VAR_INPUT
		Execute : BOOL;
		ErrorNum : DINT;
	END_VAR
	VAR_OUTPUT
		ErrorNumText : STRING[255];
		Error : BOOL;
		Done : BOOL;
	END_VAR
	VAR
		Internal : Internal_HA_SysErr_Lookup;
	END_VAR
END_FUNCTION_BLOCK

{REDUND_ERROR} FUNCTION_BLOCK HA_SysErr_Log (*Returns System Error If It Exists In Table*) (*$GROUP=User,$CAT=User,$GROUPICON=User.png,$CATICON=User.png*)
	VAR_INPUT
		Execute : BOOL;
		ErrorNum : DINT;
	END_VAR
	VAR_OUTPUT
		ErrorNumText : STRING[255];
		Error : BOOL;
		Done : BOOL;
	END_VAR
	VAR
		Internal : Internal_HA_SysErr_Log;
	END_VAR
END_FUNCTION_BLOCK
```

#### HA_SysErr_Lookup.st
```iecst
(* Returns System Error If It Exists In Table *)
FUNCTION_BLOCK HA_SysErr_Lookup

	IF NOT Execute THEN
		Internal.State := 0;
	END_IF;
	CASE Internal.State OF
		0:
			brsmemset(ADR(ErrorNumText),0,SIZEOF(ErrorNumText));
			Internal.ArTextSysGetText_0.Execute := FALSE;
			Error := FALSE;
			Done := FALSE;
			IF Execute THEN
				Internal.State := 10;
			END_IF;
		10:
			brsmemset(ADR(ErrorNumText),0,SIZEOF(ErrorNumText));
			brsmemset(ADR(Internal.TextID),0,SIZEOF(Internal.TextID));
			brsmemset(ADR(Internal.ErrorNumString),0,SIZEOF(Internal.ErrorNumString));
			brsitoa(ErrorNum,ADR(Internal.ErrorNumString));
			brsstrcat(ADR(Internal.TextID),ADR('HA_SysErr.'));
			brsstrcat(ADR(Internal.TextID),ADR(Internal.ErrorNumString));
			Internal.ArTextSysGetText_0.Execute := TRUE;
			Internal.State := 20;
		20:
			IF Internal.ArTextSysGetText_0.Done THEN
				Done := TRUE;
				Internal.State := 30;
			ELSIF Internal.ArTextSysGetText_0.Error THEN
				Error := TRUE;
				Internal.State := 30;
			END_IF;
		30:
			IF Error THEN
				ErrorNumText := 'Not Found';
			END_IF;
	END_CASE;
	Internal.ArTextSysGetText_0(Namespace := ADR('HA_SysErr'), TextID := ADR(Internal.TextID), LanguageCode := 'en', TextBufferSize := SIZEOF(ErrorNumText)-1, TextBuffer := ADR(ErrorNumText), SearchMode := arTEXTSYS_SEARCH_LANGUAGE_ONLY);

END_FUNCTION_BLOCK
```

#### HA_SysErr_Log.st
```iecst
(* Returns System Error If It Exists In Table and Logs it to the user logger*)
FUNCTION_BLOCK HA_SysErr_Log
	IF NOT Execute THEN
		Internal.State := 0;
	END_IF;
	CASE Internal.State OF
		0:
			brsmemset(ADR(ErrorNumText),0,SIZEOF(ErrorNumText));
			Internal.HA_SysErr_Lookup_0.Execute := FALSE;
			Error := FALSE;
			Done := FALSE;
			IF Execute THEN
				Internal.State := 10;
			END_IF;
		10:
			brsmemset(ADR(ErrorNumText),0,SIZEOF(ErrorNumText));
			Internal.HA_SysErr_Lookup_0.ErrorNum := ErrorNum;
			Internal.HA_SysErr_Lookup_0.Execute := TRUE;
			Internal.State := 20;
		20:
			IF Internal.HA_SysErr_Lookup_0.Done THEN
				ErrorNumText := Internal.HA_SysErr_Lookup_0.ErrorNumText;
				Internal.State := 100;
			ELSIF Internal.HA_SysErr_Lookup_0.Error THEN
				ErrorNumText := Internal.HA_SysErr_Lookup_0.ErrorNumText;
				Internal.State := 99;
			END_IF;
		99:
			Error := TRUE;
		100:
			brsmemset(ADR(Internal.AddData),0,SIZEOF(Internal.AddData));
			brsstrcat(ADR(Internal.AddData),ADR(ErrorNumText));
			Internal.ArEventLogGetIdent_0.Name := '$$arlogusr';
			Internal.ArEventLogGetIdent_0.Execute := TRUE;
			Internal.State := 110;
		110:
			IF Internal.ArEventLogGetIdent_0.Done THEN
				Internal.ArEventLogGetIdent_0.Execute := FALSE;
				Internal.ArEventLogWrite_0.Ident := Internal.ArEventLogGetIdent_0.Ident;
				Internal.ArEventLogWrite_0.EventID := -536870912;
				Internal.ArEventLogWrite_0.ObjectID := 'HA_SysErr';
				Internal.ArEventLogWrite_0.AddDataFormat := 1;
				Internal.ArEventLogWrite_0.AddData := ADR(Internal.AddData);
				Internal.ArEventLogWrite_0.AddDataSize := brsstrlen(ADR(Internal.AddData))+1;
				Internal.ArEventLogWrite_0.Execute := TRUE;
				Internal.State := 120;
			ELSIF Internal.ArEventLogGetIdent_0.Error THEN
				Internal.State := 999;
			END_IF;
		120:
			IF Internal.ArEventLogWrite_0.Done THEN
				Internal.ArEventLogWrite_0.Execute := FALSE;
				Internal.State := 130;
			ELSIF NOT Internal.ArEventLogWrite_0.Error THEN
				Internal.State := 999;
			END_IF;
		130:
			Done := TRUE;
		999:
			Error := TRUE;
			ErrorNumText := 'Log Error';
	END_CASE;
	Internal.HA_SysErr_Lookup_0();
	Internal.ArEventLogGetIdent_0();
	Internal.ArEventLogWrite_0();
END_FUNCTION_BLOCK
```

### Library Logical/Libraries/HA_Str (IEC)

#### Types.typ - Exported data types
```iecst
TYPE
	HA_brsstrcat_Internal_typ : 	STRUCT
		SrcSize : UDINT;
		DestSize : UDINT;
	END_STRUCT;
	HA_Find_Extract_Internal_typ : 	STRUCT
		i : UDINT;
		sB : UDINT;
		sSL : UDINT;
		sSR : UDINT;
		Len : UDINT;
		Pos : UDINT;
		P1 : DINT;
		P2 : DINT;
	END_STRUCT;
	HA_Find_S_Internal_typ : 	STRUCT
		i : UDINT;
		sB : UDINT;
		sS : UDINT;
	END_STRUCT;
	HA_Find_R_Internal_typ : 	STRUCT
		i : UDINT;
		sB : UDINT;
		sS : UDINT;
	END_STRUCT;
	HA_Find_L_Internal_typ : 	STRUCT
		i : UDINT;
		sB : UDINT;
		sS : UDINT;
	END_STRUCT;
END_TYPE
```

#### HA_Str.fun - Exported functions and function blocks
```iecst
FUNCTION HA_brsstrcat : BOOL
	VAR_INPUT
		pDest : UDINT;
		pSrc : UDINT;
		DestSize : UDINT;
	END_VAR
	VAR
		Internal : HA_brsstrcat_Internal_typ;
	END_VAR
END_FUNCTION

{REDUND_ERROR} FUNCTION HA_Find_L : DINT (*Returns index of substring. Negative values are Errors.*) (*$GROUP=User,$CAT=User,$GROUPICON=User.png,$CATICON=User.png*)
	VAR_INPUT
		pBuffer : UDINT;
		pSearch : UDINT;
	END_VAR
	VAR
		Internal : HA_Find_L_Internal_typ;
	END_VAR
END_FUNCTION

{REDUND_ERROR} FUNCTION HA_Find_R : DINT (*Returns right index of substring. Negative values are Errors.*) (*$GROUP=User,$CAT=User,$GROUPICON=User.png,$CATICON=User.png*)
	VAR_INPUT
		pBuffer : UDINT;
		pSearch : UDINT;
	END_VAR
	VAR
		Internal : HA_Find_R_Internal_typ;
	END_VAR
END_FUNCTION

{REDUND_ERROR} FUNCTION HA_Find_S : DINT (*Returns right index of substring. Negative values are Errors.*) (*$GROUP=User,$CAT=User,$GROUPICON=User.png,$CATICON=User.png*)
	VAR_INPUT
		pBuffer : UDINT;
		pSearch : UDINT;
	END_VAR
	VAR
		Internal : HA_Find_S_Internal_typ;
	END_VAR
END_FUNCTION

{REDUND_ERROR} FUNCTION HA_Find_Extract : DINT (*Returns end position for next search. Negative values are Errors.*) (*$GROUP=User,$CAT=User,$GROUPICON=User.png,$CATICON=User.png*)
	VAR_INPUT
		pBuffer : UDINT;
		pSearchL : UDINT;
		pSearchR : UDINT;
		pExtractADR : UDINT;
		pExtractSIZEOF : UDINT;
	END_VAR
	VAR
		Internal : HA_Find_Extract_Internal_typ;
	END_VAR
END_FUNCTION
```

#### HA_brsstrcat.st
```iecst
(* Checks the memory area before concatenating to prevent overrun. Returns false and doesnt concat if overrun is detected *)
FUNCTION HA_brsstrcat
	HA_brsstrcat 						:= TRUE;
	IF pSrc = 0 OR pDest = 0 OR DestSize = 0 THEN
		HA_brsstrcat 					:= FALSE;
	ELSE
		HA_brsstrcat					:= TRUE;
		brsmemset(ADR(Internal),0,SIZEOF(Internal));
		Internal.SrcSize := brsstrlen(pSrc);
		Internal.DestSize := brsstrlen(pDest);
		IF (Internal.SrcSize+Internal.DestSize) <= DestSize-1 THEN
			brsstrcat(pDest,pSrc);
		ELSE
			HA_brsstrcat				:= FALSE;
		END_IF;
	END_IF;
END_FUNCTION
```

#### HA_Find_S.st
```iecst
(* Returns Right index of substring, substring only returns result if found at START of buffer. Negative values are Errors. *)
FUNCTION HA_Find_S
	IF pBuffer = 0 OR pSearch = 0 THEN
		HA_Find_S	 						:= -2;
	ELSE
		Internal.sB							:= brsstrlen(pBuffer);
		Internal.sS							:= brsstrlen(pSearch);
		IF Internal.sB = 0 OR Internal.sB < Internal.sS THEN
		HA_Find_S	 						:= -3;
		END_IF;
	END_IF;
	IF HA_Find_S = 0 THEN
		HA_Find_S							:= -1;
		IF Internal.sS = 0 THEN
			HA_Find_S 						:= 0;
			RETURN;
		ELSE
			FOR Internal.i := 0 TO Internal.sB-Internal.sS DO
				IF brsmemcmp(pBuffer+Internal.i,pSearch,Internal.sS) = 0 THEN
					HA_Find_S 				:= Internal.i+Internal.sS;
					RETURN;
				ELSE
					RETURN;
				END_IF;
			END_FOR;
		END_IF;
	END_IF;
END_FUNCTION
```

#### HA_Find_L.st
```iecst
(* Returns Left index of substring. Negative values are Errors. *)
FUNCTION HA_Find_L
	IF pBuffer = 0 OR pSearch = 0 THEN
		HA_Find_L	 						:= -2;
	ELSE
		Internal.sB							:= brsstrlen(pBuffer);
		Internal.sS							:= brsstrlen(pSearch);
		IF Internal.sB = 0 OR Internal.sB < Internal.sS THEN
			HA_Find_L	 					:= -3;
		END_IF;
	END_IF;
	IF HA_Find_L = 0 THEN
		HA_Find_L							:= -1;
		IF Internal.sS = 0 THEN
			HA_Find_L 						:= 0;
			RETURN;
		ELSE
			FOR Internal.i := 0 TO Internal.sB-Internal.sS DO
				IF brsmemcmp(pBuffer+Internal.i,pSearch,Internal.sS) = 0 THEN
					HA_Find_L 				:= Internal.i;
					RETURN;
				END_IF;
			END_FOR;
		END_IF;
	END_IF;
END_FUNCTION
```
